ABB RAPID module: FSNM0399.MOD

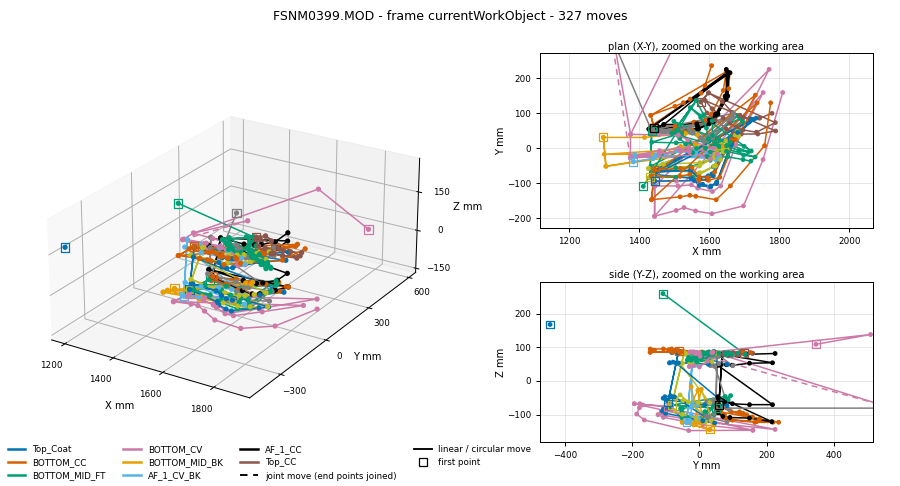
[picture p0: tool path of FSNM0399.MOD in frame currentWorkObject, 327 of 341 moves have a stored position in this frame; points joined in program order, loops and branches not executed]
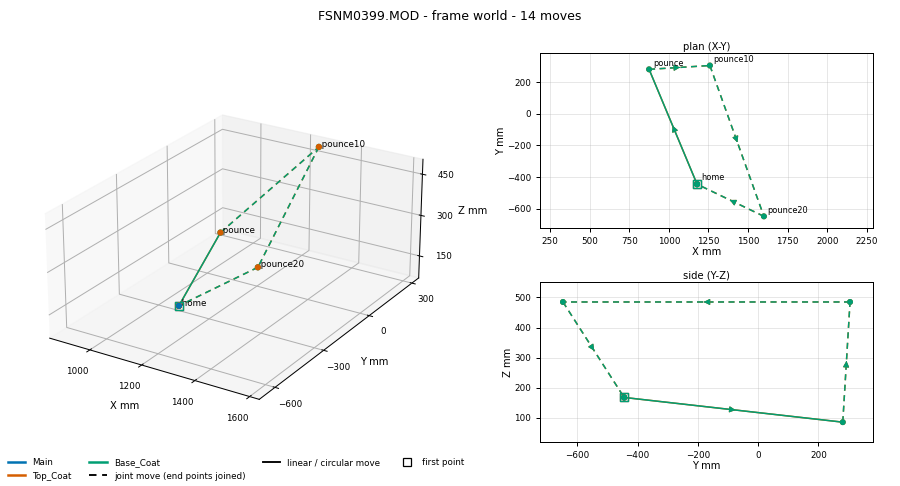
[picture p1: tool path of FSNM0399.MOD in frame world, 14 of 341 moves have a stored position in this frame; points joined in program order, loops and branches not executed]
MODULE FSNM0399
    ! 10/08/24 copied from booth 4
    !added 30 degree offset on the rotation of table to all p robtargets
    !12-02-24

    ! declare and/or define variables that are local to this module
    LOCAL CONST listitem partProgram{3}:=[[stEmpty,"Top Coat"],[stEmpty,"Flash Coat"],[stEmpty,"Stop"]];
    LOCAL VAR num itemSelected;
    LOCAL VAR btnres buttonAnswer;
    LOCAL VAR string defaultValueString;

    ! declare and/or define position variables that are local to this module
    CONST robtarget home:=[[1178.28,-445.08,168.21],[0.537841,-0.0550358,0.840932,0.0230753],[-1,0,-1,0],[-0.00413821,30.0166579,9E+09,9E+09,9E+09,9E+09]];
	CONST robtarget pounce:=[[875.08,280.72,86.17],[0.198434,0.950735,-0.173531,0.163138],[0,1,-3,1],[0.00162961,30.0303908,9E+09,9E+09,9E+09,9E+09]];
    CONST robtarget pounce2:=[[1200.4,603.09,-80.97],[0.271523,-0.961555,0.00331608,-0.0409471],[0,-1,-2,1],[-0.00391849,-6.7733,9E+09,9E+09,9E+09,9E+09]];
    CONST robtarget pounce3:=[[1412.3,-108.74,260.3],[0.92605,-0.179747,0.323715,-0.0730097],[-1,-1,-1,1],[-0.00452274,24.62897,9E+09,9E+09,9E+09,9E+09]];
    CONST robtarget pounce4:=[[1607.09,509.67,138.28],[0.628661,-0.606599,0.349538,-0.338593],[0,0,-1,1],[0.000915496,-97.692,9E+09,9E+09,9E+09,9E+09]];
    CONST robtarget pounce5:=[[1903.96,346.87,109.1],[0.946901,-0.00540743,0.281172,-0.155859],[0,0,-1,1],[-7.32737E-05,-53.436,9E+09,9E+09,9E+09,9E+09]];
    !
    ! positions for Bottom_CC (was 0)
    CONST robtarget p101:=[[1443.29,57.73,-72.18],[0.291215,0.890362,0.316501,0.149252],[0,-1,-3,1],[-0.00314945,30.0287428,9E+09,9E+09,9E+09,9E+09]];
    CONST robtarget p102:=[[1500.45,51.19,-86.06],[0.291208,0.890362,0.316527,0.14921],[0,-1,-3,1],[-0.00303958,30.0276442,9E+09,9E+09,9E+09,9E+09]];
    CONST robtarget p103:=[[1551.74,51.21,-94.97],[0.291199,0.890364,0.316549,0.149173],[0,-1,-3,1],[-0.00298465,30.0276442,9E+09,9E+09,9E+09,9E+09]];
    CONST robtarget p104:=[[1599.80,73.39,-108.74],[0.291166,0.89039,0.316497,0.149192],[0,-1,-3,1],[-0.00364383,30.0177565,9E+09,9E+09,9E+09,9E+09]];
    CONST robtarget p105:=[[1616.37,93.28,-115.08],[0.291194,0.890376,0.316552,0.149101],[0,-1,-3,1],[-0.00232547,30.0177565,9E+09,9E+09,9E+09,9E+09]];
    CONST robtarget p106:=[[1656.21,170.38,-121.36],[0.291194,0.890369,0.31654,0.149168],[0,-1,-3,1],[-0.00298465,30.0276442,9E+09,9E+09,9E+09,9E+09]];
    CONST robtarget p107:=[[1659.61,215.58,-121.43],[0.291185,0.890375,0.316546,0.149138],[0,0,-3,1],[-0.00303958,30.0287428,9E+09,9E+09,9E+09,9E+09]];

    CONST robtarget p111:=[[1433.70,63.20,-91.88],[0.0117343,-0.999087,0.013857,-0.0386828],[0,0,-2,1],[-0.00303958,30.0276442,9E+09,9E+09,9E+09,9E+09]];
    CONST robtarget p112:=[[1502.58,63.23,-91.89],[0.0117325,-0.999087,0.0138384,-0.0386773],[0,0,-2,1],[-0.00303958,30.0276442,9E+09,9E+09,9E+09,9E+09]];
    CONST robtarget p113:=[[1557.15,74.56,-101.24],[0.00782107,-0.995629,-0.0842358,-0.039561],[-1,-1,-2,1],[-0.00320438,30.0248976,9E+09,9E+09,9E+09,9E+09]];
    CONST robtarget p114:=[[1589.55,81.36,-112.17],[0.00558163,-0.989106,-0.14155,-0.0400241],[-1,-1,-2,1],[-0.00303958,30.0276442,9E+09,9E+09,9E+09,9E+09]];
    CONST robtarget p115:=[[1607.76,98.48,-116.82],[0.00228609,-0.97413,-0.222351,-0.0403144],[-1,-1,-2,1],[-0.00298465,30.0276442,9E+09,9E+09,9E+09,9E+09]];
    CONST robtarget p116:=[[1640.56,165.06,-123.31],[0.00317635,0.935526,0.350941,0.040272],[-1,-1,-2,1],[-0.00314945,30.0276442,9E+09,9E+09,9E+09,9E+09]];
    CONST robtarget p117:=[[1649.31,218.64,-123.25],[0.00148487,0.949062,0.312486,0.0404009],[-1,-1,-2,1],[-0.00314945,30.0303908,9E+09,9E+09,9E+09,9E+09]];

    CONST robtarget p121:=[[1433.69,94.12,-91.88],[0.0117298,-0.999087,0.0138599,-0.0386823],[0,0,-3,1],[-0.00314945,30.0276442,9E+09,9E+09,9E+09,9E+09]];
    CONST robtarget p122:=[[1502.66,119.56,-91.82],[0.0117433,-0.999085,0.013871,-0.0387145],[0,0,-3,1],[-0.00298465,30.0276442,9E+09,9E+09,9E+09,9E+09]];
    CONST robtarget p123:=[[1526.87,130.22,-96.62],[0.00781548,-0.995523,-0.0854657,-0.0395973],[0,-1,-2,1],[-0.0044678,30.0276442,9E+09,9E+09,9E+09,9E+09]];
    CONST robtarget p124:=[[1545.89,140.40,-100.61],[0.0049766,-0.987139,-0.154684,-0.0400532],[-1,-1,-2,1],[-0.0046326,30.0259963,9E+09,9E+09,9E+09,9E+09]];
    CONST robtarget p125:=[[1577.55,157.54,-107.21],[0.000280858,-0.962501,-0.268253,-0.0403954],[-1,-1,-2,1],[-0.00413821,30.0276442,9E+09,9E+09,9E+09,9E+09]];
    CONST robtarget p126:=[[1588.23,179.20,-113.58],[0.00322125,0.935529,0.35093,0.0402949],[-1,-1,-2,1],[-0.00303958,30.0276442,9E+09,9E+09,9E+09,9E+09]];
    CONST robtarget p127:=[[1607.33,235.84,-123.17],[0.00148313,0.949059,0.312489,0.0404348],[-1,-1,-2,1],[-0.00314945,30.0303908,9E+09,9E+09,9E+09,9E+09]];

    ! positions for Bottom_Mid_FT
    CONST robtarget p201:=[[1436.54,49.02,-81.00],[0.271519,-0.961556,0.00331699,-0.0409368],[-1,-1,-2,1],[-0.00391849,30.0276442,9E+09,9E+09,9E+09,9E+09]];
    CONST robtarget p202:=[[1505.25,48.96,-90.21],[0.271512,-0.961557,0.0033197,-0.0409763],[-1,-1,-2,1],[-0.00413821,30.0276442,9E+09,9E+09,9E+09,9E+09]];
    CONST robtarget p203:=[[1552.81,43.64,-100.76],[0.271505,-0.96156,0.00333163,-0.0409468],[-1,-1,-2,1],[-0.00413821,30.0276442,9E+09,9E+09,9E+09,9E+09]];
    CONST robtarget p204:=[[1585.76,19.14,-104.51],[0.271507,-0.96156,0.00331715,-0.0409425],[-1,-1,-2,1],[-0.00413821,30.0276442,9E+09,9E+09,9E+09,9E+09]];
    CONST robtarget p205:=[[1608.08,26.01,-109.08],[0.271524,-0.961556,0.00332285,-0.0409222],[-1,-1,-2,1],[-0.00474246,30.0375319,9E+09,9E+09,9E+09,9E+09]];
    CONST robtarget p206:=[[1682.26,92.89,-43.69],[0.402341,-0.912285,-0.052121,-0.0560508],[-1,-1,-2,1],[-0.00391849,30.0303908,9E+09,9E+09,9E+09,9E+09]];

    CONST robtarget p211:=[[1436.60,17.30,-91.94],[0.011735,-0.999088,0.013863,-0.0386529],[-1,-1,-2,1],[-0.00232547,30.0287428,9E+09,9E+09,9E+09,9E+09]];
    CONST robtarget p212:=[[1506.18,15.55,-92.02],[0.0117446,-0.999089,0.0138604,-0.0386237],[-1,-1,-2,1],[-0.00227054,30.0276442,9E+09,9E+09,9E+09,9E+09]];
    CONST robtarget p213:=[[1542.77,17.35,-103.56],[0.0117339,-0.99909,0.0138665,-0.0385899],[-1,-1,-2,1],[-0.00397342,30.0276442,9E+09,9E+09,9E+09,9E+09]];
    CONST robtarget p214:=[[1589.66,0.44,-112.40],[0.00591902,-0.990216,-0.133581,-0.039919],[-1,-1,-2,1],[-0.00413821,30.0259963,9E+09,9E+09,9E+09,9E+09]];
    CONST robtarget p215:=[[1617.25,17.02,-119.22],[0.0134057,-0.964936,-0.244424,-0.0947362],[-1,-1,-2,1],[-0.00421971,30.0124,9E+09,9E+09,9E+09,9E+09]];
    CONST robtarget p216:=[[1688.08,85.47,-55.86],[0.11425,-0.916205,-0.320136,-0.212199],[-1,-1,-2,1],[-0.00345066,30.0283,9E+09,9E+09,9E+09,9E+09]];

    CONST robtarget p221:=[[1434.12,-51.00,-82.33],[0.011678,-0.999092,0.013757,-0.0385823],[-1,-1,-2,1],[-0.0035889,30.0276442,9E+09,9E+09,9E+09,9E+09]];
    CONST robtarget p222:=[[1505.25,-56.16,-82.31],[0.0116708,-0.999092,0.0137614,-0.038585],[-1,-1,-2,1],[-0.00391849,30.0276442,9E+09,9E+09,9E+09,9E+09]];
    CONST robtarget p223:=[[1547.93,-51.91,-93.28],[0.0117018,-0.999089,0.0138091,-0.0386385],[-1,-1,-2,1],[-0.00375369,30.0276442,9E+09,9E+09,9E+09,9E+09]];
    CONST robtarget p224:=[[1603.55,-34.15,-108.91],[0.00590476,-0.990221,-0.133536,-0.0399377],[-1,-1,-2,1],[-0.00419315,30.0232497,9E+09,9E+09,9E+09,9E+09]];
    CONST robtarget p225:=[[1629.40,4.59,-115.74],[0.0150417,-0.963868,-0.24833,-0.0952052],[-1,-1,-2,1],[-0.00166629,30.0276442,9E+09,9E+09,9E+09,9E+09]];
    CONST robtarget p226:=[[1695.55,76.69,-46.30],[0.0448516,-0.904048,-0.346613,-0.246057],[-1,-1,-2,1],[-0.00430301,30.0331374,9E+09,9E+09,9E+09,9E+09]];

    CONST robtarget p231:=[[1430.77,-82.82,-71.90],[0.397779,0.811585,0.342717,0.256216],[-1,-1,-3,1],[-0.0044678,30.0259963,9E+09,9E+09,9E+09,9E+09]];
    CONST robtarget p232:=[[1505.44,-82.86,-71.95],[0.397771,0.811601,0.342711,0.256186],[-1,-1,-3,1],[-0.00452274,30.0259963,9E+09,9E+09,9E+09,9E+09]];
    CONST robtarget p233:=[[1553.31,-82.91,-84.74],[0.397775,0.811609,0.342704,0.256163],[-1,-1,-3,1],[-0.0044678,30.0259963,9E+09,9E+09,9E+09,9E+09]];
    CONST robtarget p234:=[[1612.71,-52.30,-109.68],[0.321546,0.808842,0.401441,0.285005],[-1,-1,-3,1],[-0.00562137,30.0232497,9E+09,9E+09,9E+09,9E+09]];
    CONST robtarget p235:=[[1640.12,-7.20,-117.38],[0.246617,0.798841,0.453092,0.309421],[-1,-1,-3,1],[-0.00474246,30.0248976,9E+09,9E+09,9E+09,9E+09]];
    CONST robtarget p236:=[[1684.90,48.98,-65.64],[0.201361,0.789519,0.481719,0.322583],[-1,-1,-3,1],[-0.00408328,30.0248976,9E+09,9E+09,9E+09,9E+09]];

    ! positions for Bottom_CV
    CONST robtarget p301:=[[1444.83,-93.71,-76.53],[0.271479,-0.96157,0.00322958,-0.0408855],[-1,-1,-2,1],[-0.00408328,30.0259963,9E+09,9E+09,9E+09,9E+09]];
    CONST robtarget p302:=[[1507.28,-93.73,-76.49],[0.271482,-0.961568,0.00323968,-0.0409014],[-1,-1,-2,1],[-0.00408328,30.0259963,9E+09,9E+09,9E+09,9E+09]];
    CONST robtarget p303:=[[1557.57,-92.03,-85.03],[0.271497,-0.961565,0.00327167,-0.040877],[-1,-1,-2,1],[-0.00408328,30.0259963,9E+09,9E+09,9E+09,9E+09]];
    CONST robtarget p304:=[[1571.10,-104.01,-86.44],[0.29665,-0.954764,-0.0181434,-0.00973617],[-1,-1,-2,1],[-0.00194095,30.0232497,9E+09,9E+09,9E+09,9E+09]];
    CONST robtarget p305:=[[1600.60,-111.44,-95.38],[0.382944,-0.91297,-0.0955342,0.103505],[-1,-2,-1,1],[-0.00474246,30.0248976,9E+09,9E+09,9E+09,9E+09]];
    CONST robtarget p306:=[[1621.26,-100.73,-103.16],[0.416924,-0.886981,-0.128269,0.151613],[-1,-2,-1,1],[-0.00408328,30.0259963,9E+09,9E+09,9E+09,9E+09]];
    CONST robtarget p307:=[[1663.81,10.26,-121.98],[0.425374,-0.836841,-0.276994,0.205009],[-1,-2,-1,1],[-0.00413821,30.0259963,9E+09,9E+09,9E+09,9E+09]];
    CONST robtarget p308:=[[1771.45,225.26,-144.35],[0.425406,-0.836816,-0.277007,0.205026],[-1,-2,-1,1],[-0.00430301,30.0248976,9E+09,9E+09,9E+09,9E+09]];

    CONST robtarget p311:=[[1446.22,-107.52,-79.90],[0.0862574,-0.99549,-0.0188114,-0.0347304],[-1,-1,-2,1],[-0.00633548,30.0232497,9E+09,9E+09,9E+09,9E+09]];
    CONST robtarget p312:=[[1510.91,-107.53,-79.86],[0.086252,-0.995489,-0.0188167,-0.0347533],[-1,-1,-2,1],[-0.00452274,30.0232497,9E+09,9E+09,9E+09,9E+09]];
    CONST robtarget p313:=[[1549.64,-104.32,-90.45],[0.0862414,-0.995491,-0.0187987,-0.0347426],[-1,-1,-2,1],[-0.0046326,30.0232497,9E+09,9E+09,9E+09,9E+09]];
    CONST robtarget p314:=[[1567.66,-114.11,-90.81],[0.091524,-0.993017,-0.06691,-0.0326126],[-1,-1,-2,1],[-0.00490726,30.0259963,9E+09,9E+09,9E+09,9E+09]];
    CONST robtarget p315:=[[1609.70,-123.55,-100.36],[0.116273,-0.939307,-0.322099,-0.0208838],[-1,-2,-2,1],[-0.00501712,30.0276442,9E+09,9E+09,9E+09,9E+09]];
    CONST robtarget p316:=[[1633.26,-107.63,-108.53],[0.131524,-0.897461,-0.419933,-0.0303523],[-1,-2,-2,1],[-0.0046326,30.0259963,9E+09,9E+09,9E+09,9E+09]];
    CONST robtarget p317:=[[1676.62,10.32,-130.67],[0.126766,-0.838941,-0.527221,-0.0463282],[-1,-2,-2,1],[-0.00474246,30.0259963,9E+09,9E+09,9E+09,9E+09]];
    CONST robtarget p318:=[[1754.60,159.12,-146.78],[0.126784,-0.838971,-0.527166,-0.0463555],[-1,-2,-2,1],[-0.0046326,30.0276442,9E+09,9E+09,9E+09,9E+09]];

    CONST robtarget p321:=[[1444.55,-193.95,-67.85],[0.0862284,-0.995491,-0.0189117,-0.0347111],[-1,-1,-2,1],[-0.00485233,30.0232497,9E+09,9E+09,9E+09,9E+09]];
    CONST robtarget p322:=[[1506.18,-177.54,-67.87],[0.0862406,-0.995491,-0.0188637,-0.0347006],[-1,-1,-2,1],[-0.00474246,30.0248976,9E+09,9E+09,9E+09,9E+09]];
    CONST robtarget p323:=[[1528.48,-169.22,-71.35],[0.0862428,-0.995492,-0.018788,-0.0347132],[-1,-1,-2,1],[-0.00468753,30.0232497,9E+09,9E+09,9E+09,9E+09]];
    CONST robtarget p324:=[[1561.44,-178.93,-80.05],[0.0861848,-0.995495,-0.0188292,-0.0347342],[-1,-1,-2,1],[-0.00485233,30.0232497,9E+09,9E+09,9E+09,9E+09]];
    CONST robtarget p325:=[[1608.29,-186.93,-98.69],[0.0959634,-0.975328,-0.198609,-0.009],[-1,-2,-2,1],[-0.00468753,30.0259963,9E+09,9E+09,9E+09,9E+09]];
    CONST robtarget p326:=[[1698.24,-164.47,-116.23],[0.131535,-0.89746,-0.419933,-0.0303462],[-1,-2,-2,1],[-0.00474246,30.0259963,9E+09,9E+09,9E+09,9E+09]];
    CONST robtarget p327:=[[1754.19,-32.14,-147.82],[0.12676,-0.838972,-0.527174,-0.0463151],[-1,-2,-2,1],[-0.00490726,30.0259963,9E+09,9E+09,9E+09,9E+09]];
    CONST robtarget p328:=[[1810.33,159.14,-146.82],[0.126797,-0.838964,-0.527176,-0.0463386],[-1,-2,-2,1],[-0.00468753,30.0276442,9E+09,9E+09,9E+09,9E+09]];

   ! positions for Bottom_Mid_BK (was-239)
    CONST robtarget p401:=[[1298.43,30.96,-144.46],[0.0863255,-0.995487,-0.0188879,-0.0345872],[-1,-1,-2,1],[-0.00210574,-209.559,9E+09,9E+09,9E+09,9E+09]];
    CONST robtarget p402:=[[1415.94,30.93,-144.48],[0.0863333,-0.995487,-0.0188638,-0.0345821],[-1,-1,-2,1],[-0.00216068,-209.559,9E+09,9E+09,9E+09,9E+09]];
    CONST robtarget p403:=[[1532.85,42.23,-131.08],[0.116632,-0.983288,-0.00625292,-0.139655],[-1,-1,-2,1],[-0.00243533,-209.551,9E+09,9E+09,9E+09,9E+09]];
    CONST robtarget p404:=[[1567.50,38.13,-118.46],[0.157995,-0.961788,0.00864358,-0.223441],[-1,-1,-2,1],[-0.00205081,-209.556,9E+09,9E+09,9E+09,9E+09]];
    CONST robtarget p405:=[[1640.83,5.60,-24.76],[0.0552997,-0.907428,0.181655,-0.374858],[0,0,-2,1],[-0.00270999,-209.541,9E+09,9E+09,9E+09,9E+09]];

    CONST robtarget p411:=[[1300.80,-17.20,-130.70],[0.0869689,0.992854,0.0491363,0.0652935],[0,0,-3,1],[-0.00249027,-209.554,9E+09,9E+09,9E+09,9E+09]];
    CONST robtarget p412:=[[1440.31,-17.23,-130.72],[0.0869705,0.992855,0.0491266,0.0652869],[0,0,-3,1],[-0.00243533,-209.554,9E+09,9E+09,9E+09,9E+09]];
    CONST robtarget p413:=[[1518.76,5.39,-125.44],[0.0795871,0.985904,-0.0163939,0.146255],[0,0,-3,1],[-0.00232547,-209.556,9E+09,9E+09,9E+09,9E+09]];
    CONST robtarget p414:=[[1560.70,10.21,-120.97],[0.0790598,0.972342,-0.0536054,0.213137],[0,0,-3,1],[-0.00205081,-209.555,9E+09,9E+09,9E+09,9E+09]];
    CONST robtarget p415:=[[1640.87,-4.86,-27.79],[0.0819587,0.928742,-0.0308905,0.360232],[0,0,-3,1],[-0.00265506,-209.539,9E+09,9E+09,9E+09,9E+09]];

    CONST robtarget p421:=[[1305.69,-51.36,-123.40],[0.470282,0.878825,0.0198524,0.078149],[0,0,-3,1],[-0.00260013,-209.552,9E+09,9E+09,9E+09,9E+09]];
    CONST robtarget p422:=[[1440.41,-29.26,-123.42],[0.470284,0.878824,0.0198681,0.0781488],[0,0,-3,1],[-0.00265506,-209.554,9E+09,9E+09,9E+09,9E+09]];
    CONST robtarget p423:=[[1518.27,-6.62,-120.66],[0.470322,0.878812,0.0198618,0.0780516],[0,0,-3,1],[-0.00265506,-209.554,9E+09,9E+09,9E+09,9E+09]];
    CONST robtarget p424:=[[1559.68,-3.39,-115.13],[0.45901,0.850325,0.104352,0.235305],[0,0,-3,1],[-0.00249027,-209.554,9E+09,9E+09,9E+09,9E+09]];
    CONST robtarget p425:=[[1631.23,-24.88,-17.49],[0.459095,0.850494,0.103994,0.234687],[0,0,-3,1],[-0.00249027,-209.556,9E+09,9E+09,9E+09,9E+09]];

    ! positions for AF_1_CV_BK
    CONST robtarget p501:=[[1384.21,-38.58,-123.48],[0.470286,0.878826,0.0198206,0.0781167],[0,0,-3,1],[-0.00413821,-209.552,9E+09,9E+09,9E+09,9E+09]];
    CONST robtarget p502:=[[1440.26,-29.34,-118.00],[0.470312,0.878812,0.0199042,0.0780984],[0,0,-3,1],[-0.00260013,-209.554,9E+09,9E+09,9E+09,9E+09]];
    CONST robtarget p503:=[[1515.10,-4.33,-111.47],[0.46506,0.864362,0.0727792,0.176921],[0,0,-3,1],[-0.00380863,-209.551,9E+09,9E+09,9E+09,9E+09]];
    CONST robtarget p504:=[[1559.69,-3.40,-111.67],[0.459012,0.850323,0.104336,0.235315],[0,0,-3,1],[-0.00249027,-209.555,9E+09,9E+09,9E+09,9E+09]];
    CONST robtarget p505:=[[1627.60,-25.13,-99.58],[0.597508,0.734614,0.156551,0.280745],[0,0,-3,1],[-0.00298465,-209.553,9E+09,9E+09,9E+09,9E+09]];

    CONST robtarget p511:=[[1380.35,-23.37,-78.20],[0.658363,0.746356,-0.00306919,0.0974798],[0,0,-3,1],[-0.00270999,-209.55,9E+09,9E+09,9E+09,9E+09]];
    CONST robtarget p512:=[[1446.53,-23.35,-78.18],[0.658355,0.74636,-0.00308581,0.0974916],[0,0,-3,1],[-0.00265506,-209.551,9E+09,9E+09,9E+09,9E+09]];
    CONST robtarget p513:=[[1508.74,-6.65,-72.91],[0.659338,0.731707,0.0553536,0.163748],[0,0,-3,1],[-0.00287479,-209.548,9E+09,9E+09,9E+09,9E+09]];
    CONST robtarget p514:=[[1562.72,-6.85,-66.23],[0.652837,0.704593,0.129099,0.246344],[0,0,-3,1],[-0.00298465,-209.553,9E+09,9E+09,9E+09,9E+09]];
    CONST robtarget p515:=[[1628.54,-22.53,-66.32],[0.642274,0.68584,0.174134,0.294594],[0,0,-3,1],[-0.00281986,-209.553,9E+09,9E+09,9E+09,9E+09]];

    CONST robtarget p521:=[[1380.43,-23.31,57.52],[0.658336,0.746374,-0.0031022,0.0975206],[0,0,-3,1],[-0.00265506,-209.551,9E+09,9E+09,9E+09,9E+09]];
    CONST robtarget p522:=[[1446.49,-21.21,51.74],[0.658375,0.746347,-0.00306339,0.0974654],[0,0,-3,1],[-0.00281986,-209.551,9E+09,9E+09,9E+09,9E+09]];
    CONST robtarget p523:=[[1518.33,-8.56,47.50],[0.65833,0.746377,-0.00312752,0.0975382],[0,0,-3,1],[-0.00336917,-209.547,9E+09,9E+09,9E+09,9E+09]];
    CONST robtarget p524:=[[1561.80,-13.34,47.37],[0.652819,0.704592,0.129147,0.24637],[0,0,-3,1],[-0.00298465,-209.555,9E+09,9E+09,9E+09,9E+09]];
    CONST robtarget p525:=[[1628.57,-30.08,54.41],[0.642266,0.685849,0.174127,0.294595],[0,0,-3,1],[-0.00270999,-209.553,9E+09,9E+09,9E+09,9E+09]];

    CONST robtarget p531:=[[1387.68,-18.56,85.61],[0.860289,0.500569,0.0963915,0.00646846],[0,0,-4,1],[-0.00265506,-209.551,9E+09,9E+09,9E+09,9E+09]];
    CONST robtarget p532:=[[1446.53,-18.57,82.71],[0.860293,0.50056,0.0964037,0.00646264],[0,0,-4,1],[-0.00270999,-209.551,9E+09,9E+09,9E+09,9E+09]];
    CONST robtarget p533:=[[1513.63,-6.99,78.97],[0.860828,0.490054,0.133959,0.0296148],[0,0,-4,1],[-0.00419315,-209.551,9E+09,9E+09,9E+09,9E+09]];
    CONST robtarget p534:=[[1554.41,-13.03,78.16],[0.860007,0.481305,0.162724,0.0474828],[0,0,-4,1],[-0.00260013,-209.552,9E+09,9E+09,9E+09,9E+09]];
    CONST robtarget p535:=[[1618.80,-32.62,75.28],[0.759252,0.587863,0.200244,0.194569],[0,0,-4,1],[-0.00298465,-209.557,9E+09,9E+09,9E+09,9E+09]];

    ! positions for AF_1_CC (was 0 )
    CONST robtarget p601:=[[1443.25,57.72,-72.21],[0.291214,0.890362,0.316508,0.149239],[0,-1,-3,1],[-0.00298465,30.0540114,9E+09,9E+09,9E+09,9E+09]];
    CONST robtarget p602:=[[1566.88,55.81,-95.01],[0.291153,0.890389,0.316527,0.14916],[0,-1,-3,1],[-0.00227054,30.0276442,9E+09,9E+09,9E+09,9E+09]];
    CONST robtarget p603:=[[1599.80,69.47,-105.48],[0.291161,0.89039,0.316503,0.149188],[0,-1,-3,1],[-0.0035889,30.0177565,9E+09,9E+09,9E+09,9E+09]];
    CONST robtarget p604:=[[1617.50,90.60,-108.76],[0.291202,0.890364,0.316568,0.149127],[0,-1,-3,1],[-0.00243533,30.0177565,9E+09,9E+09,9E+09,9E+09]];
    CONST robtarget p605:=[[1645.73,148.92,-110.79],[0.291203,0.890342,0.316611,0.149159],[0,-1,-3,1],[-0.00314945,30.0259963,9E+09,9E+09,9E+09,9E+09]];
    CONST robtarget p606:=[[1659.60,215.58,-121.44],[0.291184,0.890375,0.316547,0.149136],[0,0,-3,1],[-0.00298465,30.0287428,9E+09,9E+09,9E+09,9E+09]];

    CONST robtarget p611:=[[1428.47,54.73,-46.91],[0.640801,0.729046,0.164669,0.175357],[0,0,-3,1],[-0.0015015,30.0122634,9E+09,9E+09,9E+09,9E+09]];
    CONST robtarget p612:=[[1570.59,55.45,-54.72],[0.639788,0.727933,0.168626,0.179862],[0,0,-3,1],[-0.00172122,30.0166579,9E+09,9E+09,9E+09,9E+09]];
    CONST robtarget p613:=[[1612.70,75.88,-63.86],[0.588824,0.672584,0.301685,0.331517],[0,0,-3,1],[0.000311248,30.0150099,9E+09,9E+09,9E+09,9E+09]];
    CONST robtarget p614:=[[1624.95,98.15,-67.85],[0.570432,0.652282,0.335206,0.369828],[0,-1,-3,1],[-0.00188602,30.0150099,9E+09,9E+09,9E+09,9E+09]];
    CONST robtarget p615:=[[1653.26,149.10,-70.62],[0.519358,0.599464,0.427106,0.434156],[-1,-1,-4,1],[-0.00194095,30.0150099,9E+09,9E+09,9E+09,9E+09]];
    CONST robtarget p616:=[[1653.27,217.58,-70.60],[0.519357,0.599456,0.427103,0.434171],[-1,-1,-4,1],[-0.00216068,30.0166579,9E+09,9E+09,9E+09,9E+09]];

    CONST robtarget p621:=[[1428.49,54.76,46.43],[0.642228,0.730561,0.159005,0.168942],[0,0,-3,1],[-0.0015015,30.0139113,9E+09,9E+09,9E+09,9E+09]];
    CONST robtarget p622:=[[1567.14,62.93,47.45],[0.639492,0.727595,0.1698,0.181172],[0,0,-3,1],[-0.00177615,30.0150099,9E+09,9E+09,9E+09,9E+09]];
    CONST robtarget p623:=[[1608.30,80.76,48.41],[0.593251,0.677444,0.292908,0.321446],[0,0,-3,1],[0.000695769,30.0150099,9E+09,9E+09,9E+09,9E+09]];
    CONST robtarget p624:=[[1624.94,98.15,46.66],[0.570429,0.652285,0.335199,0.369833],[0,-1,-3,1],[-0.00194095,30.0139113,9E+09,9E+09,9E+09,9E+09]];
    CONST robtarget p625:=[[1653.28,149.09,52.72],[0.519362,0.599463,0.4271,0.434156],[-1,-1,-3,1],[-0.00188602,30.0150099,9E+09,9E+09,9E+09,9E+09]];
    CONST robtarget p626:=[[1653.41,217.58,54.15],[0.519362,0.59945,0.427095,0.434181],[-1,-1,-3,1],[-0.00205081,30.0166579,9E+09,9E+09,9E+09,9E+09]];

    CONST robtarget p631:=[[1470.63,67.44,79.39],[0.873611,0.349345,0.289245,0.176348],[0,0,-4,1],[-0.00188602,30.0150099,9E+09,9E+09,9E+09,9E+09]];
    CONST robtarget p632:=[[1565.05,70.05,77.01],[0.873614,0.34935,0.289207,0.176388],[0,0,-4,1],[-0.00188602,30.0150099,9E+09,9E+09,9E+09,9E+09]];
    CONST robtarget p633:=[[1601.46,80.99,78.43],[0.845134,0.335245,0.33248,0.250631],[0,-1,-4,1],[-0.0034241,30.00292498,9E+09,9E+09,9E+09,9E+09]];
    CONST robtarget p634:=[[1618.49,97.47,77.32],[0.80615,0.316649,0.376315,0.329002],[-1,-1,-4,1],[-0.00155643,30.0150099,9E+09,9E+09,9E+09,9E+09]];
    CONST robtarget p635:=[[1649.26,140.01,79.28],[0.742826,0.284916,0.420106,0.436512],[-1,-1,-4,1],[-0.00155643,30.0150099,9E+09,9E+09,9E+09,9E+09]];
    CONST robtarget p636:=[[1649.32,225.31,81.82],[0.74285,0.284897,0.420083,0.436507],[-1,-1,-4,1],[-0.00155643,30.0150099,9E+09,9E+09,9E+09,9E+09]];

    ! positions for Top_CC (was -56)

    CONST robtarget p701:=[[1576.46,132.54,82.39],[0.83287,0.421723,0.0988944,-0.344526],[0,1,-4,1],[-0.00287479,-26.1389,9E+09,9E+09,9E+09,9E+09]];
    CONST robtarget p702:=[[1594.15,100.62,82.37],[0.83285,0.421759,0.0988249,-0.344549],[0,1,-4,1],[-0.00287479,-26.1389,9E+09,9E+09,9E+09,9E+09]];
    CONST robtarget p703:=[[1617.81,81.12,77.62],[0.832842,0.421798,0.098779,-0.344534],[0,1,-4,1],[-0.00298465,-26.1213,9E+09,9E+09,9E+09,9E+09]];
    CONST robtarget p704:=[[1648.96,55.08,78.85],[0.832851,0.421766,0.0987772,-0.344553],[0,1,-4,1],[-0.00298465,-26.1235,9E+09,9E+09,9E+09,9E+09]];
    CONST robtarget p705:=[[1669.42,43.49,79.41],[0.851227,0.445293,0.118438,-0.251197],[0,0,-4,1],[-0.00281986,-26.1224,9E+09,9E+09,9E+09,9E+09]];
    CONST robtarget p706:=[[1692.05,40.47,82.03],[0.862269,0.456654,0.153412,-0.156284],[0,0,-4,1],[-0.00314945,-26.118,9E+09,9E+09,9E+09,9E+09]];
    CONST robtarget p707:=[[1739.20,40.83,84.40],[0.854107,0.464793,0.225232,0.0611466],[0,0,-4,1],[-0.00314945,-26.1246,9E+09,9E+09,9E+09,9E+09]];
    CONST robtarget p708:=[[1790.07,49.38,85.13],[0.854099,0.464806,0.225248,0.0611108],[0,0,-4,1],[-0.00270999,-26.1246,9E+09,9E+09,9E+09,9E+09]];

    CONST robtarget p711:=[[1589.13,135.98,82.41],[0.877347,0.0696564,0.239749,-0.409793],[0,0,-5,1],[-0.00287479,-26.1389,9E+09,9E+09,9E+09,9E+09]];
    CONST robtarget p712:=[[1609.04,112.91,77.33],[0.877332,0.0696555,0.23977,-0.409814],[0,0,-5,1],[-0.00303958,-26.1378,9E+09,9E+09,9E+09,9E+09]];
    CONST robtarget p713:=[[1640.79,85.92,74.73],[0.877338,0.0696414,0.239764,-0.409807],[0,0,-5,1],[-0.00281986,-26.1378,9E+09,9E+09,9E+09,9E+09]];
    CONST robtarget p714:=[[1659.83,71.33,78.37],[0.888009,0.0339087,0.256461,-0.380155],[0,0,-5,1],[-0.0034241,-26.1378,9E+09,9E+09,9E+09,9E+09]];
    CONST robtarget p715:=[[1678.62,59.81,78.21],[0.920361,0.0543184,0.259057,-0.287879],[0,0,-4,1],[-0.0044678,-26.1367,9E+09,9E+09,9E+09,9E+09]];
    CONST robtarget p716:=[[1696.78,52.22,79.48],[0.931948,0.0508699,0.262865,-0.244516],[0,0,-4,1],[-0.00435794,-26.1345,9E+09,9E+09,9E+09,9E+09]];
    CONST robtarget p717:=[[1735.36,45.89,82.98],[0.943492,0.0451952,0.265694,-0.19284],[0,0,-4,1],[-0.00419315,-26.1334,9E+09,9E+09,9E+09,9E+09]];
    CONST robtarget p718:=[[1789.23,73.30,84.33],[0.943508,0.0452016,0.265658,-0.19281],[0,0,-4,1],[-0.00419315,-26.1334,9E+09,9E+09,9E+09,9E+09]];

    CONST robtarget p721:=[[1598.70,158.11,82.46],[0.877356,0.0696883,0.239726,-0.409783],[0,0,-5,1],[-0.00287479,-26.14,9E+09,9E+09,9E+09,9E+09]];
    CONST robtarget p722:=[[1637.80,133.58,82.33],[0.877338,0.0696427,0.239777,-0.409798],[0,0,-5,1],[-0.00303958,-26.14,9E+09,9E+09,9E+09,9E+09]];
    CONST robtarget p723:=[[1665.62,102.91,78.78],[0.877352,0.0696183,0.23977,-0.409776],[0,0,-5,1],[-0.00281986,-26.1378,9E+09,9E+09,9E+09,9E+09]];
    CONST robtarget p724:=[[1688.16,94.28,82.00],[0.888022,0.0339077,0.256442,-0.380137],[0,0,-5,1],[-0.00336917,-26.1422,9E+09,9E+09,9E+09,9E+09]];
    CONST robtarget p725:=[[1698.51,88.37,81.96],[0.920358,0.0543187,0.259057,-0.287889],[0,0,-4,1],[-0.0044678,-26.1378,9E+09,9E+09,9E+09,9E+09]];
    CONST robtarget p726:=[[1715.82,84.85,82.03],[0.931958,0.050878,0.26285,-0.244491],[0,0,-4,1],[-0.00435794,-26.1356,9E+09,9E+09,9E+09,9E+09]];
    CONST robtarget p727:=[[1744.33,85.73,84.24],[0.943483,0.0451951,0.265716,-0.192852],[0,0,-4,1],[-0.00435794,-26.1323,9E+09,9E+09,9E+09,9E+09]];
    CONST robtarget p728:=[[1779.73,99.75,84.39],[0.943517,0.04522,0.265627,-0.192804],[0,0,-4,1],[-0.00430301,-26.1279,9E+09,9E+09,9E+09,9E+09]];

    ! positions for AF_1_CV_FT (was 0 )
    CONST robtarget p801:=[[1436.54,49.02,-81.00],[0.271519,-0.961556,0.00331699,-0.0409368],[-1,-1,-2,1],[-0.00391849,30.0276442,9E+09,9E+09,9E+09,9E+09]];
    CONST robtarget p802:=[[1552.88,43.61,-96.80],[0.271493,-0.961562,0.00331851,-0.0409751],[-1,-1,-2,1],[-0.00413821,30.0276442,9E+09,9E+09,9E+09,9E+09]];
    CONST robtarget p803:=[[1585.76,19.14,-104.51],[0.271507,-0.96156,0.00331715,-0.0409425],[-1,-1,-2,1],[-0.00413821,30.0276442,9E+09,9E+09,9E+09,9E+09]];
    CONST robtarget p804:=[[1610.35,28.21,-109.48],[0.271517,-0.961557,0.00331912,-0.0409256],[-1,-1,-2,1],[-0.00419315,30.0430251,9E+09,9E+09,9E+09,9E+09]];
    CONST robtarget p805:=[[1662.16,82.19,-122.39],[0.568048,-0.820114,0.0681277,-0.00962216],[-1,-1,-1,1],[-0.00397342,30.0287428,9E+09,9E+09,9E+09,9E+09]];

    CONST robtarget p811:=[[1433.92,39.75,-56.32],[0.620444,-0.728657,0.189412,-0.219614],[-1,-1,-2,1],[-0.00452274,30.0177565,9E+09,9E+09,9E+09,9E+09]];
    CONST robtarget p812:=[[1548.03,45.65,-61.28],[0.640734,-0.752133,0.101312,-0.116154],[-1,-1,-2,1],[-0.00485233,30.00567156,9E+09,9E+09,9E+09,9E+09]];
    CONST robtarget p813:=[[1595.77,21.80,-62.25],[0.643129,-0.754871,0.0848575,-0.0967134],[-1,-1,-2,1],[-0.00485233,30.0194045,9E+09,9E+09,9E+09,9E+09]];
    CONST robtarget p814:=[[1608.24,33.58,-63.93],[0.646612,-0.75881,0.0520395,-0.058245],[-1,-1,-2,1],[-0.00452274,30.0194045,9E+09,9E+09,9E+09,9E+09]];
    CONST robtarget p815:=[[1668.89,88.05,-84.84],[0.64648,-0.758638,0.0538028,-0.0603069],[-1,-1,-1,1],[-0.00474246,30.0194045,9E+09,9E+09,9E+09,9E+09]];

    CONST robtarget p821:=[[1440.49,45.86,43.15],[0.620446,-0.728662,0.189393,-0.219612],[-1,-1,-2,1],[-0.00452274,30.0177565,9E+09,9E+09,9E+09,9E+09]];
    CONST robtarget p822:=[[1543.57,57.35,51.22],[0.649961,-0.743923,0.0997815,-0.119051],[-1,-1,-2,1],[-0.00529178,30.0194045,9E+09,9E+09,9E+09,9E+09]];
    CONST robtarget p823:=[[1595.67,32.13,45.82],[0.643151,-0.75485,0.0849182,-0.0966804],[-1,-1,-2,1],[-0.00474246,30.0205031,9E+09,9E+09,9E+09,9E+09]];
    CONST robtarget p824:=[[1601.17,38.36,46.45],[0.644716,-0.756563,0.0723968,-0.0819324],[-1,-1,-2,1],[-0.00474246,30.0111647,9E+09,9E+09,9E+09,9E+09]];
    CONST robtarget p825:=[[1668.83,99.45,45.36],[0.646161,-0.758273,0.0575624,-0.0646919],[-1,-1,-1,1],[-0.00490726,30.0194045,9E+09,9E+09,9E+09,9E+09]];

    CONST robtarget p831:=[[1439.54,52.38,79.96],[0.783605,-0.54144,0.256624,-0.164167],[-1,-1,-1,1],[-0.00430301,30.0276442,9E+09,9E+09,9E+09,9E+09]];
    CONST robtarget p832:=[[1543.49,56.52,72.51],[0.7836,-0.541443,0.256617,-0.164187],[-1,-1,-1,1],[-0.00419315,30.0259963,9E+09,9E+09,9E+09,9E+09]];
    CONST robtarget p833:=[[1576.92,30.26,74.51],[0.802626,-0.574002,0.162115,0.00567045],[-1,-1,-1,1],[-0.00430301,30.0177565,9E+09,9E+09,9E+09,9E+09]];
    CONST robtarget p834:=[[1607.87,41.14,75.73],[0.802613,-0.578113,0.140663,0.0425682],[-1,-1,-1,1],[-0.00391849,30.0177565,9E+09,9E+09,9E+09,9E+09]];
    CONST robtarget p835:=[[1669.27,100.03,76.81],[0.802619,-0.578084,0.140753,0.0425392],[-1,-1,-1,1],[-0.00419315,30.0177565,9E+09,9E+09,9E+09,9E+09]];

    ! positions for AF_2_CC
    CONST robtarget p901:=[[1430.77,-82.82,-71.90],[0.397779,0.811585,0.342717,0.256216],[-1,-1,-3,1],[-0.0044678,30.0259963,9E+09,9E+09,9E+09,9E+09]];
    CONST robtarget p902:=[[1571.49,-75.48,-88.09],[0.397791,0.811597,0.342707,0.256173],[-1,-1,-3,1],[-0.00452274,30.0276442,9E+09,9E+09,9E+09,9E+09]];
    CONST robtarget p903:=[[1614.45,-51.09,-99.48],[0.321558,0.808822,0.401453,0.285031],[-1,-1,-3,1],[-0.0058411,30.0276442,9E+09,9E+09,9E+09,9E+09]];
    CONST robtarget p904:=[[1640.54,-10.12,-111.69],[0.250179,0.799419,0.450837,0.30836],[-1,-1,-3,1],[-0.00485233,30.0375319,9E+09,9E+09,9E+09,9E+09]];
    CONST robtarget p905:=[[1658.55,17.83,-121.85],[0.201335,0.78951,0.481747,0.322579],[-1,-1,-3,1],[-0.00419315,30.0259963,9E+09,9E+09,9E+09,9E+09]];
    CONST robtarget p906:=[[1684.40,34.98,-118.87],[0.289552,0.734381,0.487294,0.373348],[-1,-1,-3,1],[-0.00210574,30.0430251,9E+09,9E+09,9E+09,9E+09]];

    CONST robtarget p911:=[[1427.37,-57.56,-41.61],[0.637489,0.725508,0.177064,0.189456],[0,0,-3,1],[-0.00155643,30.0122634,9E+09,9E+09,9E+09,9E+09]];
    CONST robtarget p912:=[[1573.72,-69.72,-51.51],[0.636847,0.724789,0.17947,0.192087],[0,0,-3,1],[-0.00166629,30.0166579,9E+09,9E+09,9E+09,9E+09]];
    CONST robtarget p913:=[[1618.93,-49.56,-58.58],[0.588818,0.672599,0.301672,0.331508],[0,-1,-3,1],[0.000311248,30.0150099,9E+09,9E+09,9E+09,9E+09]];
    CONST robtarget p914:=[[1632.47,-32.90,-62.57],[0.570438,0.65231,0.33518,0.369792],[-1,-1,-3,1],[-0.00188602,30.0150099,9E+09,9E+09,9E+09,9E+09]];
    CONST robtarget p915:=[[1652.16,-3.78,-65.30],[0.519361,0.599458,0.427105,0.43416],[-1,-1,-4,1],[-0.00194095,30.0122634,9E+09,9E+09,9E+09,9E+09]];
    CONST robtarget p916:=[[1679.90,30.37,-65.44],[0.494625,0.550838,0.471765,0.478917],[-1,-1,-4,1],[-0.00194095,30.0166579,9E+09,9E+09,9E+09,9E+09]];

    CONST robtarget p921:=[[1427.39,-57.52,51.74],[0.633672,0.721662,0.189879,0.203986],[0,0,-3,1],[-0.0015015,30.0122634,9E+09,9E+09,9E+09,9E+09]];
    CONST robtarget p922:=[[1572.62,-50.64,52.60],[0.636898,0.724844,0.179233,0.191932],[0,0,-3,1],[-0.00172122,30.0166579,9E+09,9E+09,9E+09,9E+09]];
    CONST robtarget p923:=[[1612.10,-27.86,53.97],[0.58882,0.672583,0.301676,0.331535],[0,0,-3,1],[0.000311248,30.0150099,9E+09,9E+09,9E+09,9E+09]];
    CONST robtarget p924:=[[1623.84,-14.14,51.96],[0.570429,0.652285,0.335199,0.369833],[0,-1,-3,1],[-0.00194095,30.0139113,9E+09,9E+09,9E+09,9E+09]];
    CONST robtarget p925:=[[1639.97,-6.14,57.49],[0.540581,0.621543,0.391879,0.409741],[-1,-1,-4,1],[-0.00227054,30.0150099,9E+09,9E+09,9E+09,9E+09]];
    CONST robtarget p926:=[[1674.80,37.22,57.57],[0.493927,0.549724,0.482299,0.470349],[-1,-1,-3,1],[-0.00210574,30.0139113,9E+09,9E+09,9E+09,9E+09]];

    CONST robtarget p931:=[[1469.42,-45.23,84.92],[0.864048,0.379376,0.287443,0.163924],[0,0,-4,1],[-0.00177615,30.0150099,9E+09,9E+09,9E+09,9E+09]];
    CONST robtarget p932:=[[1573.56,-41.09,79.73],[0.873605,0.34934,0.289264,0.176358],[0,0,-4,1],[-0.00194095,30.0150099,9E+09,9E+09,9E+09,9E+09]];
    CONST robtarget p933:=[[1600.34,-31.32,82.70],[0.845137,0.335246,0.332479,0.250622],[-1,-1,-4,1],[-0.00336917,30.00402361,9E+09,9E+09,9E+09,9E+09]];
    CONST robtarget p934:=[[1618.66,-15.73,82.09],[0.806156,0.316677,0.376331,0.328941],[-1,-1,-4,1],[-0.00139163,30.0139113,9E+09,9E+09,9E+09,9E+09]];
    CONST robtarget p935:=[[1648.02,21.61,80.47],[0.742822,0.284929,0.420099,0.436517],[-1,-1,-4,1],[-0.00122684,30.0166579,9E+09,9E+09,9E+09,9E+09]];
    CONST robtarget p936:=[[1680.13,48.48,83.03],[0.742821,0.28498,0.420124,0.436462],[-1,-1,-4,1],[-0.0013367,30.0166579,9E+09,9E+09,9E+09,9E+09]];

   ! positions for AF_2_CV
    CONST robtarget p1001:=[[1444.85,-93.71,-61.76],[0.271475,-0.961571,0.003219,-0.0408967],[-1,-1,-2,1],[-0.00408328,30.0259963,9E+09,9E+09,9E+09,9E+09]];
    CONST robtarget p1002:=[[1557.58,-92.04,-81.52],[0.271484,-0.961569,0.00326356,-0.0408785],[-1,-1,-2,1],[-0.00408328,30.0248976,9E+09,9E+09,9E+09,9E+09]];
    CONST robtarget p1003:=[[1572.31,-106.23,-83.71],[0.29672,-0.954082,0.0021845,-0.0409951],[-1,-1,-2,1],[-0.00413821,30.0259963,9E+09,9E+09,9E+09,9E+09]];
    CONST robtarget p1004:=[[1604.55,-110.23,-89.53],[0.353528,-0.934627,-0.0197872,0.0331661],[-1,-1,-1,1],[-0.00419315,30.0259963,9E+09,9E+09,9E+09,9E+09]];
    CONST robtarget p1005:=[[1621.22,-100.73,-96.38],[0.360641,-0.915462,-0.127806,0.124636],[-1,-2,-1,1],[-0.00397342,30.0259963,9E+09,9E+09,9E+09,9E+09]];
    CONST robtarget p1006:=[[1663.78,10.27,-118.74],[0.425384,-0.836834,-0.276993,0.205018],[-1,-2,-1,1],[-0.00419315,30.0259963,9E+09,9E+09,9E+09,9E+09]];
    CONST robtarget p1007:=[[1681.22,45.13,-125.51],[0.57933,-0.78024,-0.164846,0.168607],[-1,-2,-1,1],[-0.00430301,30.0485182,9E+09,9E+09,9E+09,9E+09]];

    CONST robtarget p1011:=[[1445.88,-74.72,-47.17],[0.620444,-0.728657,0.189412,-0.219614],[-1,-1,-2,1],[-0.00452274,30.0177565,9E+09,9E+09,9E+09,9E+09]];
    CONST robtarget p1012:=[[1548.51,-85.34,-44.47],[0.639277,-0.750477,0.110106,-0.126436],[-1,-1,-2,1],[-0.00501712,30.0166579,9E+09,9E+09,9E+09,9E+09]];
    CONST robtarget p1013:=[[1581.76,-102.79,-46.89],[0.643108,-0.75533,0.0831754,-0.0947158],[-1,-1,-2,1],[-0.00501712,30.0166579,9E+09,9E+09,9E+09,9E+09]];
    CONST robtarget p1014:=[[1604.77,-108.04,-51.57],[0.646748,-0.761089,-0.0305805,0.0390479],[-1,-1,-1,1],[-0.00540164,30.0122634,9E+09,9E+09,9E+09,9E+09]];
    CONST robtarget p1015:=[[1621.96,-96.07,-56.79],[0.640297,-0.752469,-0.0985101,0.118773],[-1,-2,-1,1],[-0.00562137,30.0150099,9E+09,9E+09,9E+09,9E+09]];
    CONST robtarget p1016:=[[1664.13,15.32,-71.07],[0.608348,-0.714297,-0.222742,0.264723],[-1,-2,-1,1],[-0.00562137,30.0150099,9E+09,9E+09,9E+09,9E+09]];
    CONST robtarget p1017:=[[1720.57,82.29,-73.55],[0.626675,-0.736078,-0.164314,0.196133],[-1,-2,-1,1],[-0.00518192,30.0166579,9E+09,9E+09,9E+09,9E+09]];

    CONST robtarget p1021:=[[1445.88,-68.61,52.30],[0.620446,-0.728662,0.189393,-0.219612],[-1,-1,-2,1],[-0.00452274,30.0177565,9E+09,9E+09,9E+09,9E+09]];
    CONST robtarget p1022:=[[1546.53,-62.70,53.62],[0.633788,-0.744194,0.138203,-0.159335],[-1,-1,-2,1],[-0.00474246,30.0139113,9E+09,9E+09,9E+09,9E+09]];
    CONST robtarget p1023:=[[1574.55,-88.19,53.98],[0.643444,-0.755215,0.0825519,-0.0938923],[-1,-1,-1,1],[-0.00501712,30.0150099,9E+09,9E+09,9E+09,9E+09]];
    CONST robtarget p1024:=[[1594.89,-89.35,53.89],[0.647001,-0.760546,-0.0337541,0.0426659],[-1,-1,-1,1],[-0.00578616,30.0139113,9E+09,9E+09,9E+09,9E+09]];
    CONST robtarget p1025:=[[1612.39,-78.46,56.06],[0.640298,-0.752466,-0.0985137,0.11878],[-1,-2,-1,1],[-0.00545657,30.0150099,9E+09,9E+09,9E+09,9E+09]];
    CONST robtarget p1026:=[[1664.13,26.41,49.69],[0.609108,-0.715204,-0.220652,0.262265],[-1,-2,-1,1],[-0.00553807,30.0151,9E+09,9E+09,9E+09,9E+09]];
    CONST robtarget p1027:=[[1727.13,82.38,49.35],[0.626519,-0.73587,-0.164924,0.196899],[-1,-2,-1,1],[-0.00578616,30.0150099,9E+09,9E+09,9E+09,9E+09]];

    CONST robtarget p1031:=[[1444.93,-62.09,89.11],[0.783605,-0.54144,0.256624,-0.164167],[-1,-1,-1,1],[-0.00430301,30.0276442,9E+09,9E+09,9E+09,9E+09]];
    CONST robtarget p1032:=[[1547.65,-63.93,80.20],[0.783616,-0.541431,0.256625,-0.16414],[-1,-1,-1,1],[-0.00452274,30.0287428,9E+09,9E+09,9E+09,9E+09]];
    CONST robtarget p1033:=[[1571.58,-82.51,84.39],[0.80264,-0.573947,0.162236,0.0057333],[-1,-1,-1,1],[-0.00419315,30.0166579,9E+09,9E+09,9E+09,9E+09]];
    CONST robtarget p1034:=[[1597.43,-78.56,87.07],[0.811989,-0.57268,0.0899179,0.0680151],[-1,-1,-1,1],[-0.00430301,30.0221511,9E+09,9E+09,9E+09,9E+09]];
    CONST robtarget p1035:=[[1608.53,-72.93,86.65],[0.811193,-0.572946,0.0772463,0.0879319],[-1,-1,-1,1],[-0.00353397,30.0287428,9E+09,9E+09,9E+09,9E+09]];
    CONST robtarget p1036:=[[1659.78,24.41,79.11],[0.789397,-0.553213,-0.12754,0.233541],[-1,-1,-1,1],[-0.00339573,30.0256,9E+09,9E+09,9E+09,9E+09]];
    CONST robtarget p1037:=[[1734.35,86.07,80.41],[0.802086,-0.569524,-0.0432878,0.174433],[-1,-1,-1,1],[-0.00287479,30.0287428,9E+09,9E+09,9E+09,9E+09]];

    ! positions for TOP_CV
    CONST robtarget p1101:=[[1444.93,-62.09,89.11],[0.783605,-0.54144,0.256624,-0.164167],[-1,-1,-1,1],[-0.00430301,30.0276442,9E+09,9E+09,9E+09,9E+09]];
    CONST robtarget p1102:=[[1518.54,-57.54,85.40],[0.783453,-0.541707,0.256646,-0.163975],[-1,-1,-1,1],[-0.00501712,30.0540114,9E+09,9E+09,9E+09,9E+09]];
    CONST robtarget p1103:=[[1551.28,-55.23,85.22],[0.783611,-0.541437,0.256626,-0.164141],[-1,-1,-1,1],[-0.0044678,30.0287428,9E+09,9E+09,9E+09,9E+09]];
    CONST robtarget p1104:=[[1571.71,-81.87,89.96],[0.802621,-0.573994,0.162166,0.00567045],[-1,-1,-1,1],[-0.00419315,30.0177565,9E+09,9E+09,9E+09,9E+09]];
    CONST robtarget p1105:=[[1597.39,-83.36,90.32],[0.802812,-0.576194,0.151334,0.0243337],[-1,-1,-1,1],[-0.0044678,30.0232497,9E+09,9E+09,9E+09,9E+09]];
    CONST robtarget p1106:=[[1615.79,-68.39,91.11],[0.811205,-0.572925,0.0772617,0.0879418],[-1,-1,-1,1],[-0.0035889,30.0276442,9E+09,9E+09,9E+09,9E+09]];
    CONST robtarget p1107:=[[1663.51,24.42,84.91],[0.787021,-0.548991,-0.141484,0.243287],[-1,-1,-1,1],[-0.00353397,30.0259963,9E+09,9E+09,9E+09,9E+09]];
    CONST robtarget p1108:=[[1732.12,151.68,84.90],[0.787023,-0.548994,-0.141479,0.243278],[-1,-1,-1,1],[-0.0034241,30.0259963,9E+09,9E+09,9E+09,9E+09]];

    CONST robtarget p1111:=[[1435.66,-80.16,85.37],[0.945407,-0.158845,0.284339,0.0112061],[-1,-1,-1,1],[-0.00485233,30.0540114,9E+09,9E+09,9E+09,9E+09]];
    CONST robtarget p1112:=[[1517.26,-80.17,90.74],[0.96048,-0.15194,0.232554,0.017637],[-1,-1,-1,1],[-0.00485233,30.0540114,9E+09,9E+09,9E+09,9E+09]];
    CONST robtarget p1113:=[[1545.06,-74.51,90.69],[0.960476,-0.151937,0.232568,0.0176803],[-1,-1,-1,1],[-0.00490726,30.0540114,9E+09,9E+09,9E+09,9E+09]];
    CONST robtarget p1114:=[[1570.99,-91.43,91.80],[0.953026,-0.178065,0.217439,0.11294],[-1,-1,-1,1],[-0.00490726,30.0578566,9E+09,9E+09,9E+09,9E+09]];
    CONST robtarget p1115:=[[1598.50,-91.42,93.03],[0.934718,-0.203741,0.199028,0.212554],[-1,-1,-1,1],[-0.00474246,30.0540114,9E+09,9E+09,9E+09,9E+09]];
    CONST robtarget p1116:=[[1630.72,-82.87,95.40],[0.888914,-0.23815,0.150445,0.361224],[-1,-1,-1,1],[-0.00485233,30.05511,9E+09,9E+09,9E+09,9E+09]];
    CONST robtarget p1117:=[[1675.05,24.93,82.92],[0.823238,-0.270388,0.128925,0.482232],[-1,-1,0,1],[-0.0046326,30.0540114,9E+09,9E+09,9E+09,9E+09]];
    CONST robtarget p1118:=[[1737.12,129.88,86.51],[0.823245,-0.270377,0.128923,0.482227],[-1,-1,0,1],[-0.00468753,30.0540114,9E+09,9E+09,9E+09,9E+09]];

    CONST robtarget p1121:=[[1435.59,-146.86,85.36],[0.945403,-0.158809,0.284369,0.0112292],[-1,-1,-1,1],[-0.00485233,30.0540114,9E+09,9E+09,9E+09,9E+09]];
    CONST robtarget p1122:=[[1517.23,-138.58,90.75],[0.960482,-0.151931,0.23255,0.0176586],[-1,-1,-1,1],[-0.00485233,30.05511,9E+09,9E+09,9E+09,9E+09]];
    CONST robtarget p1123:=[[1545.11,-134.26,90.74],[0.960475,-0.151947,0.232567,0.0176831],[-1,-1,-1,1],[-0.00485233,30.0540114,9E+09,9E+09,9E+09,9E+09]];
    CONST robtarget p1124:=[[1562.20,-136.99,91.78],[0.958186,-0.164365,0.225762,0.0624085],[-1,-1,-1,1],[-0.00556644,30.0660964,9E+09,9E+09,9E+09,9E+09]];
    CONST robtarget p1125:=[[1620.49,-146.83,95.29],[0.934728,-0.203756,0.199007,0.212516],[-1,-1,-1,1],[-0.00485233,30.05511,9E+09,9E+09,9E+09,9E+09]];
    CONST robtarget p1126:=[[1661.00,-107.41,95.35],[0.888913,-0.238174,0.150427,0.361218],[-1,-1,-1,1],[-0.00490726,30.056758,9E+09,9E+09,9E+09,9E+09]];
    CONST robtarget p1127:=[[1758.49,7.38,86.45],[0.823242,-0.270313,0.128929,0.482266],[-1,-1,0,1],[-0.00468753,30.0540114,9E+09,9E+09,9E+09,9E+09]];
    CONST robtarget p1128:=[[1775.90,129.80,86.52],[0.823257,-0.270339,0.128938,0.482223],[-1,-1,0,1],[-0.00468753,30.0540114,9E+09,9E+09,9E+09,9E+09]];

    ! positions for TOP_MIDDLE_FT (was -51)
    CONST robtarget p1201:=[[1563.44,136.22,79.09],[0.588938,-0.269016,0.493537,-0.580692],[0,1,-1,1],[3.65896E-05,-21.3016,9E+09,9E+09,9E+09,9E+09]];
    CONST robtarget p1202:=[[1584.61,95.57,79.04],[0.588928,-0.269044,0.493548,-0.58068],[0,1,-1,1],[-7.32737E-05,-21.3016,9E+09,9E+09,9E+09,9E+09]];
    CONST robtarget p1203:=[[1609.12,78.56,77.59],[0.588878,-0.269104,0.493589,-0.580669],[0,1,-1,1],[3.65896E-05,-21.3005,9E+09,9E+09,9E+09,9E+09]];
    CONST robtarget p1204:=[[1610.08,36.93,78.86],[0.655635,-0.479154,0.379175,-0.443599],[0,0,-1,1],[0.000585906,-21.2889,9E+09,9E+09,9E+09,9E+09]];
    CONST robtarget p1205:=[[1630.43,23.51,80.67],[0.676285,-0.525488,0.324509,-0.40149],[0,0,-1,1],[0.000530974,-21.2906,9E+09,9E+09,9E+09,9E+09]];
    CONST robtarget p1206:=[[1660.33,16.52,80.75],[0.67293,-0.489601,0.346907,-0.432564],[0,0,-1,1],[0.000229756,-21.2872,9E+09,9E+09,9E+09,9E+09]];
    CONST robtarget p1207:=[[1700.36,5.42,64.63],[0.682218,-0.482558,0.341282,-0.430398],[0,0,-1,1],[-0.00103367,-21.2872,9E+09,9E+09,9E+09,9E+09]];
    CONST robtarget p1208:=[[1720.50,-7.72,56.17],[0.693068,-0.486875,0.325577,-0.420249],[0,0,-1,1],[-0.00130833,-21.291,9E+09,9E+09,9E+09,9E+09]];

    CONST robtarget p1211:=[[1546.62,116.02,83.37],[0.891475,0.0407577,0.265973,-0.364514],[0,0,-1,1],[0.000366179,-21.3296,9E+09,9E+09,9E+09,9E+09]];
    CONST robtarget p1212:=[[1576.13,88.43,83.35],[0.891463,0.0407337,0.265991,-0.364532],[0,0,-1,1],[0.000366179,-21.3296,9E+09,9E+09,9E+09,9E+09]];
    CONST robtarget p1213:=[[1592.57,57.56,83.35],[0.891458,0.0406935,0.266013,-0.364533],[0,0,-1,1],[0.00146481,-21.3285,9E+09,9E+09,9E+09,9E+09]];
    CONST robtarget p1214:=[[1597.93,26.80,83.08],[0.886676,0.0470431,0.281604,-0.363719],[0,0,-1,1],[0.00146481,-21.3296,9E+09,9E+09,9E+09,9E+09]];
    CONST robtarget p1215:=[[1626.48,7.19,82.97],[0.918602,0.0061386,0.289321,-0.26912],[0,0,0,1],[0.00135495,-21.3296,9E+09,9E+09,9E+09,9E+09]];
    CONST robtarget p1216:=[[1650.01,7.75,73.59],[0.925192,-0.0581398,0.331323,-0.175686],[0,0,-1,1],[0.00176784,-21.3245,9E+09,9E+09,9E+09,9E+09]];
    CONST robtarget p1217:=[[1685.24,-6.33,66.63],[0.910024,0.0138576,0.388704,-0.143431],[0,0,0,1],[-0.00064915,-21.3404,9E+09,9E+09,9E+09,9E+09]];
    CONST robtarget p1218:=[[1711.70,-10.37,61.44],[0.907164,0.0282895,0.406038,-0.106707],[0,0,0,1],[-0.00031956,-21.3443,9E+09,9E+09,9E+09,9E+09]];

    CONST robtarget p1221:=[[1499.64,77.03,83.41],[0.891435,0.040694,0.266004,-0.364596],[0,0,0,1],[0.00151974,-21.3312,9E+09,9E+09,9E+09,9E+09]];
    CONST robtarget p1222:=[[1521.56,42.53,83.37],[0.891441,0.0406534,0.266033,-0.364564],[0,0,0,1],[0.00162961,-21.3296,9E+09,9E+09,9E+09,9E+09]];
    CONST robtarget p1223:=[[1542.73,17.94,83.37],[0.891447,0.0406505,0.26604,-0.364544],[0,0,0,1],[0.00151974,-21.3285,9E+09,9E+09,9E+09,9E+09]];
    CONST robtarget p1224:=[[1564.41,-0.52,83.10],[0.891471,0.0406603,0.266028,-0.364493],[0,0,0,1],[0.00151974,-21.3296,9E+09,9E+09,9E+09,9E+09]];
    CONST robtarget p1225:=[[1603.58,-10.10,85.02],[0.917291,0.00733085,0.293455,-0.269087],[0,0,0,1],[0.00127346,-21.3322,9E+09,9E+09,9E+09,9E+09]];
    CONST robtarget p1226:=[[1649.99,-8.49,75.64],[0.928332,0.00579217,0.350782,-0.12296],[0,0,0,1],[0.00127346,-21.3322,9E+09,9E+09,9E+09,9E+09]];
    CONST robtarget p1227:=[[1698.66,-19.43,68.79],[0.920762,0.0032153,0.369124,-0.12623],[0,0,0,1],[0.00113522,-21.3274,9E+09,9E+09,9E+09,9E+09]];
    CONST robtarget p1228:=[[1731.54,-24.86,61.66],[0.906158,0.00214873,0.403566,-0.126523],[0,0,0,1],[0.00146481,-21.3323,9E+09,9E+09,9E+09,9E+09]];

    CONST robtarget p1231:=[[1494.42,42.54,88.15],[0.88187,0.462614,0.0910566,0.00112872],[0,0,0,1],[0.000366179,-21.3263,9E+09,9E+09,9E+09,9E+09]];
    CONST robtarget p1232:=[[1516.47,28.05,86.80],[0.879875,0.463455,0.104576,-0.00963777],[0,0,0,1],[0.00289304,-21.3334,9E+09,9E+09,9E+09,9E+09]];
    CONST robtarget p1233:=[[1533.15,12.32,84.10],[0.875225,0.464705,0.130771,-0.0304807],[0,0,0,1],[0.000146453,-21.3274,9E+09,9E+09,9E+09,9E+09]];
    CONST robtarget p1234:=[[1553.86,-12.35,85.18],[0.886186,0.439743,0.125215,-0.0749793],[0,0,0,1],[0.000146453,-21.3274,9E+09,9E+09,9E+09,9E+09]];
    CONST robtarget p1235:=[[1594.90,-23.45,85.04],[0.892976,0.417237,0.167559,0.0207736],[0,0,0,1],[-0.000402863,-21.3285,9E+09,9E+09,9E+09,9E+09]];
    CONST robtarget p1236:=[[1653.68,-24.38,85.14],[0.880324,0.403344,0.242349,0.060092],[0,0,0,1],[-1.8342E-05,-21.3263,9E+09,9E+09,9E+09,9E+09]];
    CONST robtarget p1237:=[[1697.22,-32.23,70.31],[0.869839,0.409506,0.255424,0.102192],[0,0,0,1],[-0.000732453,-21.2807,9E+09,9E+09,9E+09,9E+09]];
    CONST robtarget p1238:=[[1719.34,-36.55,61.99],[0.862381,0.413508,0.262838,0.127385],[0,0,0,1],[-1.8342E-05,-21.3263,9E+09,9E+09,9E+09,9E+09]];

    ! positions for Top_Middle_BK (was -239)
    CONST robtarget p1301:=[[1376.05,39.78,86.20],[0.955264,0.117853,0.2452,-0.11601],[0,0,-4,1],[0.00146481,-209.546,9E+09,9E+09,9E+09,9E+09]];
    CONST robtarget p1302:=[[1456.52,38.25,84.64],[0.955275,0.117882,0.24515,-0.115995],[0,0,-4,1],[0.000695769,-209.539,9E+09,9E+09,9E+09,9E+09]];
    CONST robtarget p1303:=[[1512.75,37.20,83.47],[0.955269,0.117879,0.245184,-0.115976],[0,0,-4,1],[0.000530974,-209.544,9E+09,9E+09,9E+09,9E+09]];
    CONST robtarget p1304:=[[1539.75,23.81,58.45],[0.943557,0.113578,0.292114,-0.107092],[0,0,-4,1],[-4.49018E-05,-209.543,9E+09,9E+09,9E+09,9E+09]];
    CONST robtarget p1305:=[[1613.58,-0.23,41.58],[0.898856,0.109452,0.416799,-0.0797264],[0,0,-4,1],[-0.000154765,-209.542,9E+09,9E+09,9E+09,9E+09]];

    CONST robtarget p1311:=[[1376.07,-21.78,86.21],[0.955267,0.117857,0.245194,-0.115993],[0,0,-4,1],[0.00151974,-209.547,9E+09,9E+09,9E+09,9E+09]];
    CONST robtarget p1312:=[[1458.68,-6.85,84.55],[0.955262,0.117861,0.245207,-0.116004],[0,0,-4,1],[0.000476043,-209.539,9E+09,9E+09,9E+09,9E+09]];
    CONST robtarget p1313:=[[1512.75,-0.22,83.46],[0.955266,0.117885,0.24519,-0.115982],[0,0,-4,1],[0.000530974,-209.544,9E+09,9E+09,9E+09,9E+09]];
    CONST robtarget p1314:=[[1541.31,2.06,73.38],[0.942284,0.12384,0.290887,-0.110221],[0,0,-4,1],[-0.000402863,-209.546,9E+09,9E+09,9E+09,9E+09]];
    CONST robtarget p1315:=[[1623.67,-16.45,45.93],[0.895082,0.13702,0.414128,-0.0924765],[0,0,-4,1],[3.65896E-05,-209.543,9E+09,9E+09,9E+09,9E+09]];

    CONST robtarget p1321:=[[1375.16,-27.50,86.19],[0.853019,0.505645,0.12624,0.0272881],[0,0,-4,1],[0.00135495,-209.534,9E+09,9E+09,9E+09,9E+09]];
    CONST robtarget p1322:=[[1457.55,-15.60,86.30],[0.853008,0.505684,0.126163,0.0272558],[0,0,-4,1],[0.00113522,-209.534,9E+09,9E+09,9E+09,9E+09]];
    CONST robtarget p1323:=[[1518.91,-7.35,81.58],[0.853008,0.505685,0.126163,0.0272703],[0,0,-4,1],[0.00130002,-209.535,9E+09,9E+09,9E+09,9E+09]];
    CONST robtarget p1324:=[[1543.79,-10.13,81.24],[0.839504,0.502337,0.194849,0.0701727],[0,0,-4,1],[0.00146481,-209.539,9E+09,9E+09,9E+09,9E+09]];
    CONST robtarget p1325:=[[1604.09,-30.27,42.76],[0.831107,0.499541,0.227045,0.0903863],[0,0,-4,1],[0.000915496,-209.536,9E+09,9E+09,9E+09,9E+09]];

    ! Varables
    !LOCAL VAR num nFlameWidth:=0;
    LOCAL VAR num preheatCycleCounter:=0;
    LOCAL VAR num coatingCycleCounter:=0;
    CONST robtarget pTest1:=[[1459.00,-171.45,-60.71],[0.537841,-0.0550356,0.840931,0.0230753],[-1,0,-1,0],[-0.00413821,0.0166579,9E+9,9E+9,9E+9,9E+9]];
    VAR extjoint extjoint1:=[9E9,9E9,9E9,9E9,9E9,9E9];
    CONST robtarget p1241:=[[1685.24,-4.80,66.69],[0.918999,-0.0345312,0.372046,-0.125819],[0,0,-1,1],[-0.000429423,-21.3377,9E+09,9E+09,9E+09,9E+09]];
    CONST robtarget p1331:=[[1285.90,545.08,-72.18],[0.291197,0.890371,0.316491,0.149257],[0,0,-3,1],[-0.00328587,30.0283,9E+09,9E+09,9E+09,9E+09]];
    CONST robtarget pounce10:=[[1259.18,304.80,485.14],[0.768187,-0.164828,0.556292,-0.270665],[0,0,-1,1],[0.00165798,30.0294,9E+09,9E+09,9E+09,9E+09]];
    CONST robtarget pounce20:=[[1600.47,-648.11,485.11],[0.768178,-0.164846,0.556301,-0.270661],[-1,0,-1,1],[0.00165798,30.0294,9E+09,9E+09,9E+09,9E+09]];

    PROC Main()
        !
        StartCycle:
        ! get part program from operator
        itemSelected:=UIListView(\Result:=buttonAnswer,\Header:="Nozzle 5000",partProgram,\Buttons:=btnOKCancel,\Icon:=iconInfo,\DefaultIndex:=1);

        IF buttonAnswer=resOK THEN
            IF itemSelected=1 THEN
                currentTool:=tMinigun_alum_ext_35mm;
                currentWorkObject:=wobj0;
                Top_Coat;
            ELSEIF itemSelected=2 THEN
                currentTool:=tMinigun_alum_ext_35mm;
                currentWorkObject:=wobj0;
                Base_Coat;
            ELSEIF itemSelected=3 THEN
                GOTO StopCycle;
            ELSEIF itemSelected=4 THEN
                GOTO StopCycle;
            ELSEIF itemSelected=5 THEN
                GOTO StopCycle;
            ELSE
                GOTO StopCycle;
            ENDIF
        ELSE
            GOTO StopCycle;
        ENDIF

        GOTO StartCycle;

        StopCycle:

        ! move to home position
        MoveL home, v800, fine, currentTool\WObj:=wobj0;
        TPErase;
        TPWrite "cut the powder and the gun";
        !
    ENDPROC

    PROC Top_Coat()
        ! move to home position
        MoveJ home, v800, fine, currentTool\WObj:=wobj0;
        !EOffsSet extjoint1;
        !EOffsOff;
        !MoveL pTest1, v800, z5, currentTool\WObj:=wobj0;
        ! TC
        ! set cycle counters
        preheatCycleCounter:=1;
        coatingCycleCounter:=10;
        !
        ! allow operator to change the number of heat cycles from the default value
        defaultValueString := "default value = " + NumtoStr(preheatCycleCounter,0);
        preheatCycleCounter := UINumEntry (\Header:="Change Heat Cycles", \MsgArray:=["How many heat cycles?", defaultValueString], \InitValue:=preheatCycleCounter, \MinValue:=preheatCycleCounter-5, \MaxValue:=preheatCycleCounter+5, \AsInteger);
        ! allow operator to change the number of coating cycles from the default value
        defaultValueString := "default value = " + NumtoStr(coatingCycleCounter,0);
        coatingCycleCounter := UINumEntry (\Header:="Change Coating Cycles", \MsgArray:=["How many coating cycles?", defaultValueString], \InitValue:=coatingCycleCounter, \MinValue:=coatingCycleCounter-10, \MaxValue:=coatingCycleCounter+10, \AsInteger);
        TPErase;
        TPWrite "start gun for preheat and press 'Cycle Start'";
        !WaitDI DI_OP_start, 1;

        ! move to start position

        WHILE preheatCycleCounter>0 DO
            !
            TPErase;
            TPWrite "number of preheat cycles remaining: "\Num:=preheatCycleCounter;
          !WaitTime 3;
          BOTTOM_CC;
          BOTTOM_MID_FT;
          BOTTOM_CV;
          BOTTOM_MID_BK;
          AF_1_CV_BK;
          AF_1_CC;
          TOP_CC;
          AF_1_CV_FT;
          AF_2_CC;
          AF_2_CV;
          TOP_CV;
          TOP_MIDDLE_FT;
          TOP_MIDDLE_BK;

            ! decrement the cycle counter
            Decr preheatCycleCounter;

            ! check for single cycle selector switch or stop cycle PB
            IF DI_Single_Cycle = 1 THEN
               GOTO End;
            ENDIF
        ENDWHILE

        ! move to home position
        MoveJ home, v800, z1, currentTool\WObj:=currentWorkObject;
        !
        TPErase;
        TPWrite "start powder feeder and press           'Cycle Start'";
        WaitDI DI_OP_start, 1;

        MoveL home, v800, z5, currentTool\WObj:=wobj0;
        !
        WHILE coatingCycleCounter>0 DO
            TPErase;
            TPWrite "number of coating cycles remaining: "\Num:=coatingCycleCounter;
           !
          BOTTOM_CC;
          BOTTOM_MID_FT;
          BOTTOM_CV;
          BOTTOM_MID_BK;
          AF_1_CV_BK;
          AF_1_CC;
          TOP_CC;
          AF_1_CV_FT;
          AF_2_CC;
          AF_2_CV;
          TOP_CV;
          TOP_MIDDLE_FT;
          TOP_MIDDLE_BK;

            ! decrement the cycle counter
            Decr coatingCycleCounter;

            ! check for single cycle selector switch or stop cycle PB
            IF DI_Single_Cycle = 1 THEN
               GOTO End;
            ENDIF
        ENDWHILE

        End:

        ! move to home position
        MoveL pounce, v800, z5, currentTool\WObj:=wobj0;
        MoveJ pounce10, v800, z5, currentTool;
        MoveJ pounce20, v800, z5, currentTool;
        MoveJ home, v800, fine, currentTool\WObj:=wobj0;

        RETURN;
    ENDPROC

    PROC Base_Coat()
        ! move to home position
        MoveL home, v800, fine, currentTool\WObj:=wobj0;
        ! BC
        ! set cycle counters
        preheatCycleCounter:=1;
        coatingCycleCounter:=5;
        !
        ! allow operator to change the number of heat cycles from the default value
        defaultValueString := "default value = " + NumtoStr(preheatCycleCounter,0);
        preheatCycleCounter := UINumEntry (\Header:="Change Heat Cycles", \MsgArray:=["How many heat cycles?", defaultValueString], \InitValue:=preheatCycleCounter, \MinValue:=preheatCycleCounter-5, \MaxValue:=preheatCycleCounter+5, \AsInteger);
        !
        ! allow operator to change the number of coating cycles from the default value
        defaultValueString := "default value = " + NumtoStr(coatingCycleCounter,0);
        coatingCycleCounter := UINumEntry (\Header:="Change Coating Cycles", \MsgArray:=["How many coating cycles?", defaultValueString], \InitValue:=coatingCycleCounter, \MinValue:=coatingCycleCounter-10, \MaxValue:=coatingCycleCounter+10, \AsInteger);
        !
        TPErase;
        TPWrite "start gun for preheat and press         'Cycle Start'";
        WaitDI DI_OP_start, 1;
        !
        WHILE preheatCycleCounter>0 DO
            !
            TPErase;
            TPWrite "number of preheat cycles remaining: "\Num:=preheatCycleCounter;
            !WaitTime 4;
          BOTTOM_CC;
          BOTTOM_MID_FT;
          BOTTOM_CV;
          BOTTOM_MID_BK;
          AF_1_CV_BK;
          AF_1_CC;
          TOP_CC;
          AF_1_CV_FT;
          AF_2_CC;
          AF_2_CV;
          TOP_CV;
          TOP_MIDDLE_FT;
          TOP_MIDDLE_BK;
          !
            ! decrement the cycle counter
            Decr preheatCycleCounter;

            ! check for single cycle selector switch or stop cycle PB
            IF DI_Single_Cycle = 1 THEN
               GOTO End;
            ENDIF
        ENDWHILE

        ! move to pounce position
        MoveJ home, v800, fine, currentTool\WObj:=wobj0;
        !
        TPErase;
        TPWrite "start powder feeder and press 'Cycle Start'";
        WaitDI DI_OP_start, 1;
        MoveL home, v800, z5, currentTool\WObj:=wobj0;
        !
        WHILE coatingCycleCounter>0 DO
            TPErase;
            TPWrite "number of coating cycles remaining: "\Num:=coatingCycleCounter;
           !
           !WaitTime 4;
          BOTTOM_CC;
          BOTTOM_MID_FT;
          BOTTOM_CV;
          BOTTOM_MID_BK;
          AF_1_CV_BK;
          AF_1_CC;
          TOP_CC;
          AF_1_CV_FT;
          AF_2_CC;
          AF_2_CV;
          TOP_CV;
          TOP_MIDDLE_FT;
          TOP_MIDDLE_BK;

            ! decrement the cycle counter
            Decr coatingCycleCounter;

            ! check for single cycle selector switch or stop cycle PB
            IF DI_Single_Cycle = 1 THEN
               GOTO End;
            ENDIF
        ENDWHILE

        End:

        ! move to home position
        MoveL pounce, v800, z5, currentTool\WObj:=wobj0;
        MoveJ pounce10, v800, z5, currentTool;
        MoveJ pounce20, v800, z5, currentTool;
        MoveJ home, v800, fine, currentTool\WObj:=wobj0;

        RETURN;
    ENDPROC

    PROC BOTTOM_CC()
        currentpath := z30;
        !
        MoveJ p101, v800, z1, currentTool\WObj:=currentWorkObject;
        !
        ! Radius
        SpeedFactors_3 0.8, .6, .7, .5, .5, .6, .8, 1, 1, 1;
        SpeedFactors_4 .6, .6, .5, .5, .6, .8, 1, 1, 1, 1;
        Para2 2, 400, 101, 111, 7, 0.0;
        !
        ! Flat
        SpeedFactors_3 .3, .4, .4, 6, .4, .5, 1, 1, 1, 1;
        SpeedFactors_4 .4, .3, 6, .4, .5, 1, 1, 1, 1, 1;
        Para2 2, 600, 111, 121, 7, 0.0;
        !
        MoveL p121, v800, z1, currentTool\WObj:=currentWorkObject;
        !
        RETURN;
        MoveL p101, v500, z1, currentTool\WObj:=currentWorkObject;
        MoveL p102, v500, z1, currentTool\WObj:=currentWorkObject;
        MoveL p103, v500, z1, currentTool\WObj:=currentWorkObject;
        MoveL p104, v500, z1, currentTool\WObj:=currentWorkObject;
        MoveL p105, v500, z1, currentTool\WObj:=currentWorkObject;
        MoveL p106, v500, z1, currentTool\WObj:=currentWorkObject;
        MoveL p107, v500, z1, currentTool\WObj:=currentWorkObject;
        !
        MoveL p111, v500, z1, currentTool\WObj:=currentWorkObject;
        MoveL p112, v500, z1, currentTool\WObj:=currentWorkObject;
        MoveL p113, v500, z1, currentTool\WObj:=currentWorkObject;
        MoveL p114, v500, z1, currentTool\WObj:=currentWorkObject;
        MoveL p115, v500, z1, currentTool\WObj:=currentWorkObject;
        MoveL p116, v500, z1, currentTool\WObj:=currentWorkObject;
        MoveL p117, v500, z1, currentTool\WObj:=currentWorkObject;
        !
        MoveL p121, v500, z1, currentTool\WObj:=currentWorkObject;
        MoveL p122, v500, z1, currentTool\WObj:=currentWorkObject;
        MoveL p123, v500, z1, currentTool\WObj:=currentWorkObject;
        MoveL p124, v500, z1, currentTool\WObj:=currentWorkObject;
        MoveL p125, v500, z1, currentTool\WObj:=currentWorkObject;
        MoveL p126, v500, z1, currentTool\WObj:=currentWorkObject;
        MoveL p127, v500, z1, currentTool\WObj:=currentWorkObject;
        !

    ENDPROC

    PROC BOTTOM_MID_FT()
        currentpath := z30;
        !
        MoveL p201, v800, z1, currentTool\WObj:=currentWorkObject;
        !
        ! Left Radius
        SpeedFactors_3 1, 1, 1.3, 1.5, .9, 3, 1, 1, 1, 1;
        SpeedFactors_4 1, 1.3, 1.5, .9, 3, 1, 1, 1, 1, 1;
        Para2 2, 300, 201, 211, 6, 0.0;
        !
        ! Mid
        SpeedFactors_3 1, 1, .7, .9, 8, 8, 1, 1, 1, 1;
        SpeedFactors_4 1, .8, .8, 8, 8, 1, 1, 1, 1, 1;
        Para2 2, 350, 211, 221, 6, 0.0;
        !
        ! Right Radius
        SpeedFactors_3 1, .9, .7, .7, .6, 4, 1, 1, 1, 1;
        SpeedFactors_4 .9, .7, .7, .6, 4, 1, 1, 1, 1, 1;
        Para2 2, 300, 221, 231, 6, 0.0;
        !
        MoveL p231, v800, z1, currentTool\WObj:=currentWorkObject;
        !
        RETURN;
        MoveL p201, v500, z1, currentTool\WObj:=currentWorkObject;
        MoveL p202, v500, z1, currentTool\WObj:=currentWorkObject;
        MoveL p203, v500, z1, currentTool\WObj:=currentWorkObject;
        MoveL p204, v500, z1, currentTool\WObj:=currentWorkObject;
        MoveL p205, v500, z1, currentTool\WObj:=currentWorkObject;
        MoveL p206, v500, z1, currentTool\WObj:=currentWorkObject;
        !
        MoveL p211, v500, z1, currentTool\WObj:=currentWorkObject;
        MoveL p212, v500, z1, currentTool\WObj:=currentWorkObject;
        MoveL p213, v500, z1, currentTool\WObj:=currentWorkObject;
        MoveL p214, v500, z1, currentTool\WObj:=currentWorkObject;
        MoveL p215, v500, z1, currentTool\WObj:=currentWorkObject;
        MoveL p216, v500, z1, currentTool\WObj:=currentWorkObject;
        !
        MoveL p221, v500, z1, currentTool\WObj:=currentWorkObject;
        MoveL p222, v500, z1, currentTool\WObj:=currentWorkObject;
        MoveL p223, v500, z1, currentTool\WObj:=currentWorkObject;
        MoveL p224, v500, z1, currentTool\WObj:=currentWorkObject;
        MoveL p225, v500, z1, currentTool\WObj:=currentWorkObject;
        MoveL p226, v500, z1, currentTool\WObj:=currentWorkObject;
        !
        MoveL p231, v500, z1, currentTool\WObj:=currentWorkObject;
        MoveL p232, v500, z1, currentTool\WObj:=currentWorkObject;
        MoveL p233, v500, z1, currentTool\WObj:=currentWorkObject;
        MoveL p234, v500, z1, currentTool\WObj:=currentWorkObject;
        MoveL p235, v500, z1, currentTool\WObj:=currentWorkObject;
        MoveL p236, v500, z1, currentTool\WObj:=currentWorkObject;
        !

    ENDPROC

    PROC BOTTOM_CV()
        currentpath := z30;
        !
        MoveL p301, v800, z1, currentTool\WObj:=currentWorkObject;
        !
        ! Radius
        SpeedFactors_3 0.5, .9, .8, 9, 8, 3.5, .3, 1.1, 1, 1;
        SpeedFactors_4 .9, .8, 9, 8, 3.5, .3, 1.1, 1, 1, 1;
        Para2 2, 600, 301, 311, 8, 0.0;
        !
        ! Flat
        SpeedFactors_3 1, 1, .4, .9, 5, .7, .4, .5, 1, 1;
        SpeedFactors_4 1, .4, .9, 5, .7, .3, .5, 1, 1, 1;
        Para2 2, 600, 311, 321, 8, 0.0;
        !
        MoveL p321, v800, z1, currentTool\WObj:=currentWorkObject;
        !
        RETURN;
        MoveL p301, v500, z1, currentTool\WObj:=currentWorkObject;
        MoveL p302, v500, z1, currentTool\WObj:=currentWorkObject;
        MoveL p303, v500, z1, currentTool\WObj:=currentWorkObject;
        MoveL p304, v500, z1, currentTool\WObj:=currentWorkObject;
        MoveL p305, v500, z1, currentTool\WObj:=currentWorkObject;
        MoveL p306, v500, z1, currentTool\WObj:=currentWorkObject;
        MoveL p307, v500, z1, currentTool\WObj:=currentWorkObject;
        MoveL p308, v500, z1, currentTool\WObj:=currentWorkObject;
        !
        MoveL p311, v500, z1, currentTool\WObj:=currentWorkObject;
        MoveL p312, v500, z1, currentTool\WObj:=currentWorkObject;
        MoveL p313, v500, z1, currentTool\WObj:=currentWorkObject;
        MoveL p314, v500, z1, currentTool\WObj:=currentWorkObject;
        MoveL p315, v500, z1, currentTool\WObj:=currentWorkObject;
        MoveL p316, v500, z1, currentTool\WObj:=currentWorkObject;
        MoveL p317, v500, z1, currentTool\WObj:=currentWorkObject;
        MoveL p318, v500, z1, currentTool\WObj:=currentWorkObject;
        !
        MoveL p321, v500, z1, currentTool\WObj:=currentWorkObject;
        MoveL p322, v500, z1, currentTool\WObj:=currentWorkObject;
        MoveL p323, v500, z1, currentTool\WObj:=currentWorkObject;
        MoveL p324, v500, z1, currentTool\WObj:=currentWorkObject;
        MoveL p325, v500, z1, currentTool\WObj:=currentWorkObject;
        MoveL p326, v500, z1, currentTool\WObj:=currentWorkObject;
        MoveL p327, v500, z1, currentTool\WObj:=currentWorkObject;
        MoveL p328, v500, z1, currentTool\WObj:=currentWorkObject;
        !

    ENDPROC

    PROC BOTTOM_MID_BK()
        currentpath := z10;
        !
        MoveL p401, v800, z1, currentTool\WObj:=currentWorkObject;
        !
        ! Flat
        SpeedFactors_3 1, .4, .5, 2.8, 4, 1, 1, 1, 1, 1;
        SpeedFactors_4 .5, .5, 2.8, 4, 1, 1, 1, 1, 1, 1;
        Para2 2, 600, 401, 411, 5, 0.0;
        !
        ! Right Radius
        SpeedFactors_3 1, .9, 1.5, 1.7, 2, 1, 1, 1, 1, 1;
        SpeedFactors_4 1.3, 1.5, 1.7, 2, 1, 1, 1, 1, 1, 1;
        Para2 2, 300, 411, 421, 5, 0.0;
        !
        MoveL p421, v800, z1, currentTool\WObj:=currentWorkObject;
        !
        RETURN;
        MoveL p401, v500, z1, currentTool\WObj:=currentWorkObject;
        MoveL p402, v500, z1, currentTool\WObj:=currentWorkObject;
        MoveL p403, v500, z1, currentTool\WObj:=currentWorkObject;
        MoveL p404, v500, z1, currentTool\WObj:=currentWorkObject;
        MoveL p405, v500, z1, currentTool\WObj:=currentWorkObject;
        !
        MoveL p411, v500, z1, currentTool\WObj:=currentWorkObject;
        MoveL p412, v500, z1, currentTool\WObj:=currentWorkObject;
        MoveL p413, v500, z1, currentTool\WObj:=currentWorkObject;
        MoveL p414, v500, z1, currentTool\WObj:=currentWorkObject;
        MoveL p415, v500, z1, currentTool\WObj:=currentWorkObject;
        !
        MoveL p421, v500, z1, currentTool\WObj:=currentWorkObject;
        MoveL p422, v500, z1, currentTool\WObj:=currentWorkObject;
        MoveL p423, v500, z1, currentTool\WObj:=currentWorkObject;
        MoveL p424, v500, z1, currentTool\WObj:=currentWorkObject;
        MoveL p425, v500, z1, currentTool\WObj:=currentWorkObject;
        !
    ENDPROC

    PROC AF_1_CV_BK()
        currentpath := z40;

        MoveJ p501, v800, z1, currentTool\WObj:=currentWorkObject;
        !
        ! Bottom Radius
        SpeedFactors_3 1, 1, 1, 4, 6, 1, 1, 1, 1, 1;
        SpeedFactors_4 1, 1, 4, 6, 1, 1, 1, 1, 1, 1;
        Para2 2, 500, 501, 511, 5, 0.0;
        !
        ! Mid
        SpeedFactors_3 1, 1, .5, 6, 6, 1, 1, 1, 1, 1;
        SpeedFactors_4 1, 1, 6, 6, 1, 1, 1, 1, 1, 1;
        Para2 2, 500, 511, 521, 5, 0.0;
        !
        ! Top Radius
        SpeedFactors_3 1, 1, .5, 6, 6, 1, 1, 1, 1, 1;
        SpeedFactors_4 1, .5, 6, 6, 1, 1, 1, 1, 1, 1;
        Para2 2, 300, 521, 531, 5, 0.0;

        MoveL p531, v800, z1, currentTool\WObj:=currentWorkObject;
        !
        RETURN;
        MoveL p501, v500, z1, currentTool\WObj:=currentWorkObject;
        MoveL p502, v500, z1, currentTool\WObj:=currentWorkObject;
        MoveL p503, v500, z1, currentTool\WObj:=currentWorkObject;
        MoveL p504, v500, z1, currentTool\WObj:=currentWorkObject;
        MoveL p505, v500, z1, currentTool\WObj:=currentWorkObject;
        !
        MoveL p511, v500, z1, currentTool\WObj:=currentWorkObject;
        MoveL p512, v500, z1, currentTool\WObj:=currentWorkObject;
        MoveL p513, v500, z1, currentTool\WObj:=currentWorkObject;
        MoveL p514, v500, z1, currentTool\WObj:=currentWorkObject;
        MoveL p515, v500, z1, currentTool\WObj:=currentWorkObject;
        !
        MoveL p521, v500, z1, currentTool\WObj:=currentWorkObject;
        MoveL p522, v500, z1, currentTool\WObj:=currentWorkObject;
        MoveL p523, v500, z1, currentTool\WObj:=currentWorkObject;
        MoveL p524, v500, z1, currentTool\WObj:=currentWorkObject;
        MoveL p525, v500, z1, currentTool\WObj:=currentWorkObject;
        !
        MoveL p531, v500, z1, currentTool\WObj:=currentWorkObject;
        MoveL p532, v500, z1, currentTool\WObj:=currentWorkObject;
        MoveL p533, v500, z1, currentTool\WObj:=currentWorkObject;
        MoveL p534, v500, z1, currentTool\WObj:=currentWorkObject;
        MoveL p535, v500, z1, currentTool\WObj:=currentWorkObject;
        !
    ENDPROC

    PROC AF_1_CC()

        currentpath := z20;
        !
        MoveL p601, v800, z1, currentTool\WObj:=currentWorkObject;
        !
        ! Bottom Radius
        SpeedFactors_3 1, .2, .3, .3, .3, .3, .3, 1, 1, 1;
        SpeedFactors_4 .2, .3, .4, .3, .3, .3, 1, 1, 1, 1;
        Para2 2, 650, 601, 611, 6, 0.0;
        !
        ! Mid
        SpeedFactors_3 1, .3, .6, 1.1, .3, .3, .7, 1, 1, 1;
        SpeedFactors_4 .3, .6, 1.1, .3, .4, .7, 1, 1, 1, 1;
        Para2 2, 650, 611, 621, 6, 0.0;
        !
        ! Top Radius
        SpeedFactors_3 1, .3, .3, 1.3, .7, .4, .3, 1, 1, 1;
        SpeedFactors_4 .3, .3, 1.3, .7, .3, .3, 1, 1, 1, 1;
        Para2 2, 442, 621, 631, 6, 0.0;
        !
        MoveL p631, v800, z1, currentTool\WObj:=currentWorkObject;
        !
        RETURN;
        MoveL p601, v500, z1, currentTool\WObj:=currentWorkObject;
        MoveL p602, v500, z1, currentTool\WObj:=currentWorkObject;
        MoveL p603, v500, z1, currentTool\WObj:=currentWorkObject;
        MoveL p604, v500, z1, currentTool\WObj:=currentWorkObject;
        MoveL p605, v500, z1, currentTool\WObj:=currentWorkObject;
        MoveL p606, v500, z1, currentTool\WObj:=currentWorkObject;
        !
        MoveL p611, v500, z1, currentTool\WObj:=currentWorkObject;
        MoveL p612, v500, z1, currentTool\WObj:=currentWorkObject;
        MoveL p613, v500, z1, currentTool\WObj:=currentWorkObject;
        MoveL p614, v500, z1, currentTool\WObj:=currentWorkObject;
        MoveL p615, v500, z1, currentTool\WObj:=currentWorkObject;
        MoveL p616, v500, z1, currentTool\WObj:=currentWorkObject;
        !
        MoveL p621, v500, z1, currentTool\WObj:=currentWorkObject;
        MoveL p622, v500, z1, currentTool\WObj:=currentWorkObject;
        MoveL p623, v500, z1, currentTool\WObj:=currentWorkObject;
        MoveL p624, v500, z1, currentTool\WObj:=currentWorkObject;
        MoveL p625, v500, z1, currentTool\WObj:=currentWorkObject;
        MoveL p626, v500, z1, currentTool\WObj:=currentWorkObject;
        !
        MoveL p631, v500, z1, currentTool\WObj:=currentWorkObject;
        MoveL p632, v500, z1, currentTool\WObj:=currentWorkObject;
        MoveL p633, v500, z1, currentTool\WObj:=currentWorkObject;
        MoveL p634, v500, z1, currentTool\WObj:=currentWorkObject;
        MoveL p635, v500, z1, currentTool\WObj:=currentWorkObject;
        MoveL p636, v500, z1, currentTool\WObj:=currentWorkObject;
        !
    ENDPROC

    PROC Top_CC()

        currentpath := z40;
        !
        MoveL p701, v800, z1, currentTool\WObj:=currentWorkObject;
        !
        ! Right Radius
        SpeedFactors_3 1, 1, .4, .4, .9, .3, 1.2, 1.8, 1, 1;
        SpeedFactors_4 1, .5, .5, .9, .3, 1.2, 1.7, 1, 1, 1;
        Para2 2, 500, 701, 711, 8, 0.0;
        !
        ! Flat
        SpeedFactors_3 1, 1, .4, 6, 1.8, .8, .4, 1.8, 1, 1;
        SpeedFactors_4 1, .4, 6, 1.8, .8, .4, 1.8, 1, 1, 1;
        Para2 2, 500, 711, 721, 8, 0.0;
        !
        MoveL p721, v800, z1, currentTool\WObj:=currentWorkObject;
        !
        RETURN;
        MoveL p701, v500, z1, currentTool\WObj:=currentWorkObject;
        MoveL p702, v500, z1, currentTool\WObj:=currentWorkObject;
        MoveL p703, v500, z1, currentTool\WObj:=currentWorkObject;
        MoveL p704, v500, z1, currentTool\WObj:=currentWorkObject;
        MoveL p705, v500, z1, currentTool\WObj:=currentWorkObject;
        MoveL p706, v500, z1, currentTool\WObj:=currentWorkObject;
        MoveL p707, v500, z1, currentTool\WObj:=currentWorkObject;
        MoveL p708, v500, z1, currentTool\WObj:=currentWorkObject;
        !
        MoveL p711, v500, z1, currentTool\WObj:=currentWorkObject;
        MoveL p712, v500, z1, currentTool\WObj:=currentWorkObject;
        MoveL p713, v500, z1, currentTool\WObj:=currentWorkObject;
        MoveL p714, v500, z1, currentTool\WObj:=currentWorkObject;
        MoveL p715, v500, z1, currentTool\WObj:=currentWorkObject;
        MoveL p716, v500, z1, currentTool\WObj:=currentWorkObject;
        MoveL p717, v500, z1, currentTool\WObj:=currentWorkObject;
        MoveL p718, v500, z1, currentTool\WObj:=currentWorkObject;
        !
        MoveL p721, v500, z1, currentTool\WObj:=currentWorkObject;
        MoveL p722, v500, z1, currentTool\WObj:=currentWorkObject;
        MoveL p723, v500, z1, currentTool\WObj:=currentWorkObject;
        MoveL p724, v500, z1, currentTool\WObj:=currentWorkObject;
        MoveL p725, v500, z1, currentTool\WObj:=currentWorkObject;
        MoveL p726, v500, z1, currentTool\WObj:=currentWorkObject;
        MoveL p727, v500, z1, currentTool\WObj:=currentWorkObject;
        MoveL p728, v500, z1, currentTool\WObj:=currentWorkObject;
        !

    ENDPROC

    PROC AF_1_CV_FT()
        currentpath := z40;
        !
        MoveL pounce2, v800, z1, currentTool\WObj:=currentWorkObject;
        MoveL p801, v800, z1, currentTool\WObj:=currentWorkObject;
        !
        ! Bottom Radius
        SpeedFactors_3 1, 1, .2, .8, 6, 1, 1, 1, 1, 1;
        SpeedFactors_4 1, .2, .8, 6, 1, 1, 1, 1, 1, 1;
        Para2 2, 425, 801, 811, 5, 0.0;
        !
        ! Mid
        SpeedFactors_3 1, 1, 1.3, 3, 6, 1, 1, 1, 1, 1;
        SpeedFactors_4 1, 1.2, 3, 6, 1, 1, 1, 1, 1, 1;
        Para2 2, 475, 811, 821, 5, 0.0;
        !
        ! Top Radius
        SpeedFactors_3 1, 1, 1.3, 2, 6, 1, 1, 1, 1, 1;
        SpeedFactors_4 1, 1.3, 2, 6, 1, 1, 1, 1, 1, 1;
        Para2 2, 475, 821, 831, 5, 0.0;
        !
        MoveL p831, v800, z1, currentTool\WObj:=currentWorkObject;
        !
        RETURN;
        MoveL p801, v500, z1, currentTool\WObj:=currentWorkObject;
        MoveL p802, v500, z1, currentTool\WObj:=currentWorkObject;
        MoveL p803, v500, z1, currentTool\WObj:=currentWorkObject;
        MoveL p804, v500, z1, currentTool\WObj:=currentWorkObject;
        MoveL p805, v500, z1, currentTool\WObj:=currentWorkObject;
        !
        MoveL p811, v500, z1, currentTool\WObj:=currentWorkObject;
        MoveL p812, v500, z1, currentTool\WObj:=currentWorkObject;
        MoveL p813, v500, z1, currentTool\WObj:=currentWorkObject;
        MoveL p814, v500, z1, currentTool\WObj:=currentWorkObject;
        MoveL p815, v500, z1, currentTool\WObj:=currentWorkObject;
        !
        MoveL p821, v500, z1, currentTool\WObj:=currentWorkObject;
        MoveL p822, v500, z1, currentTool\WObj:=currentWorkObject;
        MoveL p823, v500, z1, currentTool\WObj:=currentWorkObject;
        MoveL p824, v500, z1, currentTool\WObj:=currentWorkObject;
        MoveL p825, v500, z1, currentTool\WObj:=currentWorkObject;
        !
        MoveL p831, v500, z1, currentTool\WObj:=currentWorkObject;
        MoveL p832, v500, z1, currentTool\WObj:=currentWorkObject;
        MoveL p833, v500, z1, currentTool\WObj:=currentWorkObject;
        MoveL p834, v500, z1, currentTool\WObj:=currentWorkObject;
        MoveL p835, v500, z1, currentTool\WObj:=currentWorkObject;
        !
    ENDPROC

    PROC AF_2_CC()
        currentpath := z40;
        !
        MoveL p901, v800, z1, currentTool\WObj:=currentWorkObject;
        !
        ! Bottom Radius
        SpeedFactors_3 1, .4, .5, .7, .9, 3, 1, 1, 1, 1;
        SpeedFactors_4 .4, .5, .7, .9, 3, 1, 1, 1, 1, 1;
        Para2 2, 300, 901, 911, 6, 0.0;
        !
        ! Mid
        SpeedFactors_3 1, .5, .7, .8, .4, 2, 1, 1, 1, 1;
        SpeedFactors_4 .5, .8, .8, .4, 2, 1, 1, 1, 1, 1;
        Para2 2, 300, 911, 921, 6, 0.0;
        !
        ! Top Radius
        SpeedFactors_3 1, .7, 2, .5, 3, 2.5, 1, 1, 1, 1;
        SpeedFactors_4 .7, 2.1, .5, 3, 2.5, 1, 1, 1, 1, 1;
        Para2 2, 300, 921, 931, 6, 0.0;
        !
        MoveL p931, v800, z1, currentTool\WObj:=currentWorkObject;
        !
        RETURN;
        MoveL p901, v500, z1, currentTool\WObj:=currentWorkObject;
        MoveL p902, v500, z1, currentTool\WObj:=currentWorkObject;
        MoveL p903, v500, z1, currentTool\WObj:=currentWorkObject;
        MoveL p904, v500, z1, currentTool\WObj:=currentWorkObject;
        MoveL p905, v500, z1, currentTool\WObj:=currentWorkObject;
        MoveL p906, v500, z1, currentTool\WObj:=currentWorkObject;
        !
        MoveL p911, v500, z1, currentTool\WObj:=currentWorkObject;
        MoveL p912, v500, z1, currentTool\WObj:=currentWorkObject;
        MoveL p913, v500, z1, currentTool\WObj:=currentWorkObject;
        MoveL p914, v500, z1, currentTool\WObj:=currentWorkObject;
        MoveL p915, v500, z1, currentTool\WObj:=currentWorkObject;
        MoveL p916, v500, z1, currentTool\WObj:=currentWorkObject;
        !
        MoveL p921, v500, z1, currentTool\WObj:=currentWorkObject;
        MoveL p922, v500, z1, currentTool\WObj:=currentWorkObject;
        MoveL p923, v500, z1, currentTool\WObj:=currentWorkObject;
        MoveL p924, v500, z1, currentTool\WObj:=currentWorkObject;
        MoveL p925, v500, z1, currentTool\WObj:=currentWorkObject;
        MoveL p926, v500, z1, currentTool\WObj:=currentWorkObject;
        !
        MoveL p931, v500, z1, currentTool\WObj:=currentWorkObject;
        MoveL p932, v500, z1, currentTool\WObj:=currentWorkObject;
        MoveL p933, v500, z1, currentTool\WObj:=currentWorkObject;
        MoveL p934, v500, z1, currentTool\WObj:=currentWorkObject;
        MoveL p935, v500, z1, currentTool\WObj:=currentWorkObject;
        MoveL p936, v500, z1, currentTool\WObj:=currentWorkObject;
        !
    ENDPROC

    PROC AF_2_CV()
        currentpath := z40;
        !
        MoveL p1001, v800, z1, currentTool\WObj:=currentWorkObject;
        !
        ! Bottom Radius
        SpeedFactors_3 1, 1, .2, 1.9, 8, .3, 4, 1, 1, 1;
        SpeedFactors_4 1, .2, 1.9, 8, .3, 4, 1, 1, 1, 1;
        Para2 2, 475, 1001, 1011, 7, 0.0;
        !
        ! Flat
        SpeedFactors_3 1, 1, .2, 7, 7, .3, 4, 1, 1, 1;
        SpeedFactors_4 1, .3, 7, 7, .4, 4, 1, 1, 1, 1;
        Para2 2, 475, 1011, 1021, 7, 0.0;
        !
        ! Top Radius
        SpeedFactors_3 1, 1, .6, .8, .7, .3, 4, 1, 1, 1;
        SpeedFactors_4 1, .6, .9, .7, .2, 4, 1, 1, 1, 1;
        Para2 2, 475, 1021, 1031, 7, 0.0;
        !
        MoveL p1031, v800, z1, currentTool\WObj:=currentWorkObject;
        !
        RETURN;
        MoveL p1001, v500, z1, currentTool\WObj:=currentWorkObject;
        MoveL p1002, v500, z1, currentTool\WObj:=currentWorkObject;
        MoveL p1003, v500, z1, currentTool\WObj:=currentWorkObject;
        MoveL p1004, v500, z1, currentTool\WObj:=currentWorkObject;
        MoveL p1005, v500, z1, currentTool\WObj:=currentWorkObject;
        MoveL p1006, v500, z1, currentTool\WObj:=currentWorkObject;
        MoveL p1007, v500, z1, currentTool\WObj:=currentWorkObject;
        !
        MoveL p1011, v500, z1, currentTool\WObj:=currentWorkObject;
        MoveL p1012, v500, z1, currentTool\WObj:=currentWorkObject;
        MoveL p1013, v500, z1, currentTool\WObj:=currentWorkObject;
        MoveL p1014, v500, z1, currentTool\WObj:=currentWorkObject;
        MoveL p1015, v500, z1, currentTool\WObj:=currentWorkObject;
        MoveL p1016, v500, z1, currentTool\WObj:=currentWorkObject;
        MoveL p1017, v500, z1, currentTool\WObj:=currentWorkObject;
        !
        MoveL p1021, v500, z1, currentTool\WObj:=currentWorkObject;
        MoveL p1022, v500, z1, currentTool\WObj:=currentWorkObject;
        MoveL p1023, v500, z1, currentTool\WObj:=currentWorkObject;
        MoveL p1024, v500, z1, currentTool\WObj:=currentWorkObject;
        MoveL p1025, v500, z1, currentTool\WObj:=currentWorkObject;
        MoveL p1026, v500, z1, currentTool\WObj:=currentWorkObject;
        MoveL p1027, v500, z1, currentTool\WObj:=currentWorkObject;
        !
        MoveL p1031, v500, z1, currentTool\WObj:=currentWorkObject;
        MoveL p1032, v500, z1, currentTool\WObj:=currentWorkObject;
        MoveL p1033, v500, z1, currentTool\WObj:=currentWorkObject;
        MoveL p1034, v500, z1, currentTool\WObj:=currentWorkObject;
        MoveL p1035, v500, z1, currentTool\WObj:=currentWorkObject;
        MoveL p1036, v500, z1, currentTool\WObj:=currentWorkObject;
        MoveL p1037, v500, z1, currentTool\WObj:=currentWorkObject;
        !
    ENDPROC

    PROC TOP_CV()
        currentpath := z60;
        !
        MoveL p1101, v800, z1, currentTool\WObj:=currentWorkObject;
        !
        ! Left Radius
        SpeedFactors_3 1, 1, .5, 4.5, 8, 2, .4, 1.7, 1, 1;
        SpeedFactors_4 1, .5, 4.5, 8, 2, .4, 2, 1.7, 1, 1;
        Para2 2, 500, 1101, 1111, 8, 0.0;
        !
        ! Flat
        SpeedFactors_3 1, 1, .6, .7, 5, 3, .3, .4, 1, 1;
        SpeedFactors_4 1, .6, .7, 5, 3, .4, .5, 1, 1, 1;
        Para2 2, 500, 1111, 1121, 8, 0.0;
        !
        MoveL p1121, v800, z1, currentTool\WObj:=currentWorkObject;
        !
        RETURN;
        MoveL p1101, v500, z1, currentTool\WObj:=currentWorkObject;
        MoveL p1102, v500, z1, currentTool\WObj:=currentWorkObject;
        MoveL p1103, v500, z1, currentTool\WObj:=currentWorkObject;
        MoveL p1104, v500, z1, currentTool\WObj:=currentWorkObject;
        MoveL p1105, v500, z1, currentTool\WObj:=currentWorkObject;
        MoveL p1106, v500, z1, currentTool\WObj:=currentWorkObject;
        MoveL p1107, v500, z1, currentTool\WObj:=currentWorkObject;
        MoveL p1108, v500, z1, currentTool\WObj:=currentWorkObject;
        !
        MoveL p1111, v500, z1, currentTool\WObj:=currentWorkObject;
        MoveL p1112, v500, z1, currentTool\WObj:=currentWorkObject;
        MoveL p1113, v500, z1, currentTool\WObj:=currentWorkObject;
        MoveL p1114, v500, z1, currentTool\WObj:=currentWorkObject;
        MoveL p1115, v500, z1, currentTool\WObj:=currentWorkObject;
        MoveL p1116, v500, z1, currentTool\WObj:=currentWorkObject;
        MoveL p1117, v500, z1, currentTool\WObj:=currentWorkObject;
        MoveL p1118, v500, z1, currentTool\WObj:=currentWorkObject;
        !
        MoveL p1121, v500, z1, currentTool\WObj:=currentWorkObject;
        MoveL p1122, v500, z1, currentTool\WObj:=currentWorkObject;
        MoveL p1123, v500, z1, currentTool\WObj:=currentWorkObject;
        MoveL p1124, v500, z1, currentTool\WObj:=currentWorkObject;
        MoveL p1125, v500, z1, currentTool\WObj:=currentWorkObject;
        MoveL p1126, v500, z1, currentTool\WObj:=currentWorkObject;
        MoveL p1127, v500, z1, currentTool\WObj:=currentWorkObject;
        MoveL p1128, v500, z1, currentTool\WObj:=currentWorkObject;
        !
    ENDPROC

    PROC TOP_MIDDLE_FT()
        currentpath := z30;
        !
        MoveL pounce3, v800, z1, currentTool\WObj:=currentWorkObject;
        MoveL p1201, v800, z1, currentTool\WObj:=currentWorkObject;
        !
        ! Left Radius
        SpeedFactors_3 1, 1, 1, 2, .9, 1.8, 6, 6, 1, 1;
        SpeedFactors_4 1, 1, 2, .9, 1.8, 6, 6, 1, 1, 1;
        Para2 2, 700, 1201, 1211, 8, 0.0;
        !
        ! Mid
        SpeedFactors_3 1, 1, .4, .9, 6, 6, 6, 6, 1, 1;
        SpeedFactors_4 1, .3, .9, 6, 6, 6, 6, 1, 1, 1;
        Para2 2, 700, 1211, 1221, 8, 0.0;
        !
        ! Right Radius
        SpeedFactors_3 1, 1, .7, .6, .6, 1.5, 6, 6, 1, 1;
        SpeedFactors_4 1, .7, .6, .6, 1.5, 6, 6, 1, 1, 1;
        Para2 2, 700, 1221, 1231, 8, 0.0;
        !
        MoveL p1231, v800, z1, currentTool\WObj:=currentWorkObject;
        !
        RETURN;
        !MoveL p1241, v800, z1, currentTool\WObj:=currentWorkObject;
        MoveL p1201, v500, z1, currentTool\WObj:=currentWorkObject;
        MoveL p1202, v500, z1, currentTool\WObj:=currentWorkObject;
        MoveL p1203, v500, z1, currentTool\WObj:=currentWorkObject;
        MoveL p1204, v500, z1, currentTool\WObj:=currentWorkObject;
        MoveL p1205, v500, z1, currentTool\WObj:=currentWorkObject;
        MoveL p1206, v500, z1, currentTool\WObj:=currentWorkObject;
        MoveL p1207, v500, z1, currentTool\WObj:=currentWorkObject;
        MoveL p1208, v500, z1, currentTool\WObj:=currentWorkObject;
        !
        MoveL p1211, v500, z1, currentTool\WObj:=currentWorkObject;
        MoveL p1212, v500, z1, currentTool\WObj:=currentWorkObject;
        MoveL p1213, v500, z1, currentTool\WObj:=currentWorkObject;
        MoveL p1214, v500, z1, currentTool\WObj:=currentWorkObject;
        MoveL p1215, v500, z1, currentTool\WObj:=currentWorkObject;
        MoveL p1216, v500, z1, currentTool\WObj:=currentWorkObject;
        MoveL p1217, v500, z1, currentTool\WObj:=currentWorkObject;
        MoveL p1218, v500, z1, currentTool\WObj:=currentWorkObject;
        !
        MoveL p1221, v500, z1, currentTool\WObj:=currentWorkObject;
        MoveL p1222, v500, z1, currentTool\WObj:=currentWorkObject;
        MoveL p1223, v500, z1, currentTool\WObj:=currentWorkObject;
        MoveL p1224, v500, z1, currentTool\WObj:=currentWorkObject;
        MoveL p1225, v500, z1, currentTool\WObj:=currentWorkObject;
        MoveL p1226, v500, z1, currentTool\WObj:=currentWorkObject;
        MoveL p1227, v500, z1, currentTool\WObj:=currentWorkObject;
        MoveL p1228, v500, z1, currentTool\WObj:=currentWorkObject;
        !
        MoveL p1231, v500, z1, currentTool\WObj:=currentWorkObject;
        MoveL p1232, v500, z1, currentTool\WObj:=currentWorkObject;
        MoveL p1233, v500, z1, currentTool\WObj:=currentWorkObject;
        MoveL p1234, v500, z1, currentTool\WObj:=currentWorkObject;
        MoveL p1235, v500, z1, currentTool\WObj:=currentWorkObject;
        MoveL p1236, v500, z1, currentTool\WObj:=currentWorkObject;
        MoveL p1237, v500, z1, currentTool\WObj:=currentWorkObject;
        MoveL p1238, v500, z1, currentTool\WObj:=currentWorkObject;
        !
    ENDPROC

    PROC TOP_MIDDLE_BK()
        currentpath := z30;
        !
        MoveL pounce5, v800, z1, currentTool\WObj:=currentWorkObject;
        MoveL pounce4, v800, z1, currentTool\WObj:=currentWorkObject;
        MoveL p1301, v800, z1, currentTool\WObj:=currentWorkObject;
        !
        ! Flat
        SpeedFactors_3 1, .3, .5, 6, 6, 1, 1, 1, 1, 1;
        SpeedFactors_4 .3, .5, 6, 6, 1, 1, 1, 1, 1, 1;
        Para2 2, 700, 1301, 1311, 5, 0.0;
        !
        ! Right Radius
        SpeedFactors_3 1, .8, .6, 3.5, 6, 1, 1, 1, 1, 1;
        SpeedFactors_4 .8, .6, 3.5, 6, 1, 1, 1, 1, 1, 1;
        Para2 2, 700, 1311, 1321, 5, 0.0;
        !
        MoveL p1321, v800, z1, currentTool\WObj:=currentWorkObject;
        MoveJ p1331, v800, z1, currentTool\WObj:=currentWorkObject;
        !
        RETURN;
        MoveL p1301, v500, z1, currentTool\WObj:=currentWorkObject;
        MoveL p1302, v500, z1, currentTool\WObj:=currentWorkObject;
        MoveL p1303, v500, z1, currentTool\WObj:=currentWorkObject;
        MoveL p1304, v500, z1, currentTool\WObj:=currentWorkObject;
        MoveL p1305, v500, z1, currentTool\WObj:=currentWorkObject;
        !
        MoveL p1311, v500, z1, currentTool\WObj:=currentWorkObject;
        MoveL p1312, v500, z1, currentTool\WObj:=currentWorkObject;
        MoveL p1313, v500, z1, currentTool\WObj:=currentWorkObject;
        MoveL p1314, v500, z1, currentTool\WObj:=currentWorkObject;
        MoveL p1315, v500, z1, currentTool\WObj:=currentWorkObject;
        !
        MoveL p1321, v500, z1, currentTool\WObj:=currentWorkObject;
        MoveL p1322, v500, z1, currentTool\WObj:=currentWorkObject;
        MoveL p1323, v500, z1, currentTool\WObj:=currentWorkObject;
        MoveL p1324, v500, z1, currentTool\WObj:=currentWorkObject;
        MoveL p1325, v500, z1, currentTool\WObj:=currentWorkObject;
        !
    ENDPROC
ENDMODULE
